LIN {X 0,Y 523.335,Z 404.353,A -85,B 0,C 180,E1 -4767.691,E2 -4767.691} C_VEL
LIN {X 0,Y 523.256,Z 405.957,A -85,B 0,C 180,E1 -4769.23,E2 -4769.23} C_VEL
LIN {X 0,Y 523.257,Z 406.174,A -85,B 0,C 180,E1 -4770,E2 -4770} C_VEL
LIN {X 0,Y 523.275,Z 405.351,A -85,B 0,C 180,E1 -4771.539,E2 -4771.539} C_VEL
LIN {X 0,Y 523.335,Z 404.357,A -85,B 0,C 180,E1 -4772.309,E2 -4772.309} C_VEL
LIN {X 0,Y 523.367,Z 402.961,A -85,B 0,C 180,E1 -4773.079,E2 -4773.079} C_VEL
LIN {X 0,Y 523.422,Z 400.024,A -85,B 0,C 180,E1 -4774.235,E2 -4774.235} C_VEL
LIN {X 0,Y 523.455,Z 396.045,A -85,B 0,C 180,E1 -4775.392,E2 -4775.392} C_VEL
LIN {X 0,Y 523.507,Z 389.976,A -85,B 0,C 180,E1 -4776.736,E2 -4776.736} C_VEL
LIN {X 0,Y 523.643,Z 383.242,A -85,B 0,C 180,E1 -4777.907,E2 -4777.907} C_VEL
LIN {X 0,Y 523.826,Z 374.948,A -85,B 0,C 180,E1 -4779.07,E2 -4779.07} C_VEL
LIN {X 0,Y 524.03,Z 366.449,A -85,B 0,C 180,E1 -4780.04,E2 -4780.04} C_VEL
LIN {X 0,Y 524.307,Z 355.951,A -85,B 0,C 180,E1 -4781.011,E2 -4781.011} C_VEL
LIN {X 0,Y 524.58,Z 345.751,A -85,B 0,C 180,E1 -4781.776,E2 -4781.776} C_VEL
LIN {X 0,Y 524.893,Z 334.187,A -85,B 0,C 180,E1 -4782.468,E2 -4782.468} C_VEL
LIN {X 0,Y 525.134,Z 322.52,A -85,B 0,C 180,E1 -4783.003,E2 -4783.003} C_VEL
LIN {X 0,Y 525.347,Z 309.079,A -85,B 0,C 180,E1 -4783.44,E2 -4783.44} C_VEL
LIN {X 0,Y 525.596,Z 295.824,A -85,B 0,C 180,E1 -4783.705,E2 -4783.705} C_VEL
LIN {X 0,Y 525.799,Z 203.654,A -85,B 0,C 180,E1 -4784.971,E2 -4784.971} C_VEL
LIN {X 0,Y 524.231,Z 193.19,A -85,B 0,C 180,E1 -4785.176,E2 -4785.176} C_VEL
LIN {X 0,Y 524.601,Z 174.823,A -85,B 0,C 180,E1 -4787.977,E2 -4787.977} C_VEL
LIN {X 0,Y 525.054,Z 155.376,A -85,B 0,C 180,E1 -4790.98,E2 -4790.98} C_VEL
LIN {X 0,Y 525.297,Z 140.922,A -85,B 0,C 180,E1 -4793.245,E2 -4793.245} C_VEL
LIN {X 0,Y 523.934,Z 133.223,A -85,B 0,C 180,E1 -4794.571,E2 -4794.571} C_VEL
LIN {X 0,Y 523.918,Z 133.225,A -85,B 0,C 180,E1 -4797.706,E2 -4797.706} C_VEL
LIN {X 0,Y 523.941,Z 133.217,A -85,B 0,C 180,E1 -4800.644,E2 -4800.644} C_VEL
LIN {X 0,Y 523.923,Z 133.224,A -85,B 0,C 180,E1 -4803.728,E2 -4803.728} C_VEL
LIN {X 0,Y 523.893,Z 133.222,A -85,B 0,C 180,E1 -4806.399,E2 -4806.399} C_VEL
LIN {X 0,Y 523.913,Z 133.224,A -85,B 0,C 180,E1 -4809.084,E2 -4809.084} C_VEL
LIN {X 0,Y 523.906,Z 133.22,A -85,B 0,C 180,E1 -4812.122,E2 -4812.122} C_VEL
LIN {X 0,Y 523.932,Z 133.224,A -85,B 0,C 180,E1 -4815.31,E2 -4815.31} C_VEL
LIN {X 0,Y 523.913,Z 133.222,A -85,B 0,C 180,E1 -4818.694,E2 -4818.694} C_VEL
LIN {X 0,Y 523.904,Z 133.22,A -85,B 0,C 180,E1 -4821.897,E2 -4821.897} C_VEL
LIN {X 0,Y 523.909,Z 133.228,A -85,B 0,C 180,E1 -4824.912,E2 -4824.912} C_VEL
LIN {X 0,Y 523.922,Z 133.218,A -85,B 0,C 180,E1 -4827.68,E2 -4827.68} C_VEL
LIN {X 0,Y 523.926,Z 133.225,A -85,B 0,C 180,E1 -4830.68,E2 -4830.68} C_VEL
LIN {X 0,Y 523.893,Z 133.222,A -85,B 0,C 180,E1 -4833.724,E2 -4833.724} C_VEL
LIN {X 0,Y 523.895,Z 133.225,A -85,B 0,C 180,E1 -4836.269,E2 -4836.269} C_VEL
LIN {X 0,Y 523.919,Z 133.224,A -85,B 0,C 180,E1 -4838.765,E2 -4838.765} C_VEL
LIN {X 0,Y 523.914,Z 133.22,A -85,B 0,C 180,E1 -4841.219,E2 -4841.219} C_VEL
LIN {X 0,Y 523.899,Z 133.229,A -85,B 0,C 180,E1 -4844.437,E2 -4844.437} C_VEL
LIN {X 0,Y 523.934,Z 133.217,A -85,B 0,C 180,E1 -4847.607,E2 -4847.607} C_VEL
LIN {X 0,Y 523.933,Z 133.219,A -85,B 0,C 180,E1 -4850.737,E2 -4850.737} C_VEL
LIN {X 0,Y 523.99,Z 133.214,A -85,B 0,C 180,E1 -4853.84,E2 -4853.84} C_VEL
LIN {X 0,Y 524.093,Z 133.201,A -85,B 0,C 180,E1 -4857.694,E2 -4857.694} C_VEL
LIN {X 0,Y 524.086,Z 133.206,A -85,B 0,C 180,E1 -4860,E2 -4860} C_VEL
LIN {X 0,Y 524.094,Z 133.2,A -85,B 0,C 180,E1 -4862.306,E2 -4862.306} C_VEL
LIN {X 0,Y 523.999,Z 133.212,A -85,B 0,C 180,E1 -4866.16,E2 -4866.16} C_VEL
LIN {X 0,Y 523.968,Z 133.215,A -85,B 0,C 180,E1 -4869.262,E2 -4869.262} C_VEL
LIN {X 0,Y 523.987,Z 133.218,A -85,B 0,C 180,E1 -4871.736,E2 -4871.736} C_VEL
LIN {X 0,Y 523.973,Z 133.214,A -85,B 0,C 180,E1 -4875.049,E2 -4875.049} C_VEL
LIN {X 0,Y 523.903,Z 133.223,A -85,B 0,C 180,E1 -4877.971,E2 -4877.971} C_VEL
LIN {X 0,Y 523.942,Z 133.215,A -85,B 0,C 180,E1 -4880.411,E2 -4880.411} C_VEL
LIN {X 0,Y 523.897,Z 133.224,A -85,B 0,C 180,E1 -4882.894,E2 -4882.894} C_VEL
LIN {X 0,Y 523.89,Z 133.229,A -85,B 0,C 180,E1 -4885.422,E2 -4885.422} C_VEL
LIN {X 0,Y 523.897,Z 133.221,A -85,B 0,C 180,E1 -4888.003,E2 -4888.003} C_VEL
LIN {X 0,Y 523.926,Z 133.223,A -85,B 0,C 180,E1 -4890.853,E2 -4890.853} C_VEL
LIN {X 0,Y 523.922,Z 133.219,A -85,B 0,C 180,E1 -4893.73,E2 -4893.73} C_VEL
LIN {X 0,Y 523.895,Z 133.223,A -85,B 0,C 180,E1 -4896.402,E2 -4896.402} C_VEL
LIN {X 0,Y 523.905,Z 133.226,A -85,B 0,C 180,E1 -4899.086,E2 -4899.086} C_VEL
LIN {X 0,Y 523.902,Z 133.221,A -85,B 0,C 180,E1 -4902.124,E2 -4902.124} C_VEL
LIN {X 0,Y 523.935,Z 133.218,A -85,B 0,C 180,E1 -4905.311,E2 -4905.311} C_VEL
LIN {X 0,Y 523.895,Z 133.227,A -85,B 0,C 180,E1 -4906.872,E2 -4906.872} C_VEL
LIN {X 0,Y 523.223,Z 133.308,A -85,B 0,C 180,E1 -4907.513,E2 -4907.513} C_VEL
LIN {X 0,Y 520.362,Z 133.67,A -85,B 0,C 180,E1 -4908.555,E2 -4908.555} C_VEL
LIN {X 0,Y 517.955,Z 133.965,A -85,B 0,C 180,E1 -4909.393,E2 -4909.393} C_VEL
LIN {X 0,Y 516.935,Z 134.091,A -85,B 0,C 180,E1 -4910.041,E2 -4910.041} C_VEL
LIN {X 0,Y 516.859,Z 134.102,A -85,B 0,C 180,E1 -4910.261,E2 -4910.261} C_VEL
LIN {X 0,Y 516.85,Z 134.099,A -85,B 0,C 180,E1 -4913.253,E2 -4913.253} C_VEL
LIN {X 0,Y 516.904,Z 134.097,A -85,B 0,C 180,E1 -4916.121,E2 -4916.121} C_VEL
LIN {X 0,Y 516.886,Z 134.096,A -85,B 0,C 180,E1 -4918.937,E2 -4918.937} C_VEL
LIN {X 0,Y 516.85,Z 134.1,A -85,B 0,C 180,E1 -4921.582,E2 -4921.582} C_VEL
LIN {X 0,Y 516.877,Z 134.104,A -85,B 0,C 180,E1 -4924.209,E2 -4924.209} C_VEL
LIN {X 0,Y 516.857,Z 134.099,A -85,B 0,C 180,E1 -4926.777,E2 -4926.777} C_VEL
LIN {X 0,Y 516.968,Z 134.097,A -85,B 0,C 180,E1 -4930.132,E2 -4930.132} C_VEL
LIN {X 0,Y 517.566,Z 139.303,A -85,B 0,C 180,E1 -4931.187,E2 -4931.187} C_VEL
LIN {X 0,Y 517.249,Z 154.128,A -85,B 0,C 180,E1 -4934.03,E2 -4934.03} C_VEL
LIN {X 0,Y 517.253,Z 157.604,A -85,B 0,C 180,E1 -4934.68,E2 -4934.68} C_VEL
LIN {X 0,Y 519.135,Z 167.747,A -85,B 0,C 180,E1 -4934.89,E2 -4934.89} C_VEL
LIN {X 0,Y 518.683,Z 264.861,A -85,B 0,C 180,E1 -4936.259,E2 -4936.259} C_VEL
LIN {X 0,Y 518.509,Z 278.018,A -85,B 0,C 180,E1 -4936.604,E2 -4936.604} C_VEL
LIN {X 0,Y 518.244,Z 291.213,A -85,B 0,C 180,E1 -4937.121,E2 -4937.121} C_VEL
LIN {X 0,Y 517.973,Z 303.019,A -85,B 0,C 180,E1 -4937.757,E2 -4937.757} C_VEL
LIN {X 0,Y 517.715,Z 314.443,A -85,B 0,C 180,E1 -4938.549,E2 -4938.549} C_VEL
LIN {X 0,Y 517.401,Z 324.683,A -85,B 0,C 180,E1 -4939.434,E2 -4939.434} C_VEL
LIN {X 0,Y 517.114,Z 333.868,A -85,B 0,C 180,E1 -4940.417,E2 -4940.417} C_VEL
LIN {X 0,Y 516.821,Z 342.781,A -85,B 0,C 180,E1 -4941.595,E2 -4941.595} C_VEL
LIN {X 0,Y 516.621,Z 349.955,A -85,B 0,C 180,E1 -4942.772,E2 -4942.772} C_VEL
LIN {X 0,Y 516.511,Z 356.489,A -85,B 0,C 180,E1 -4944.143,E2 -4944.143} C_VEL
LIN {X 0,Y 516.351,Z 360.813,A -85,B 0,C 180,E1 -4945.316,E2 -4945.316} C_VEL
LIN {X 0,Y 516.378,Z 363.097,A -85,B 0,C 180,E1 -4946.098,E2 -4946.098} C_VEL
LIN {X 0,Y 516.353,Z 364.958,A -85,B 0,C 180,E1 -4946.88,E2 -4946.88} C_VEL
LIN {X 0,Y 516.267,Z 366.366,A -85,B 0,C 180,E1 -4947.66,E2 -4947.66} C_VEL
LIN {X 0,Y 516.17,Z 367.982,A -85,B 0,C 180,E1 -4949.22,E2 -4949.22} C_VEL
LIN {X 0,Y 516.167,Z 368.219,A -85,B 0,C 180,E1 -4950,E2 -4950} C_VEL
LIN {X 0,Y 516.17,Z 368.036,A -85,B 0,C 180,E1 -4950.781,E2 -4950.781} C_VEL
LIN {X 0,Y 516.267,Z 366.49,A -85,B 0,C 180,E1 -4952.341,E2 -4952.341} C_VEL
LIN {X 0,Y 516.354,Z 365.137,A -85,B 0,C 180,E1 -4953.121,E2 -4953.121} C_VEL
LIN {X 0,Y 516.394,Z 362.28,A -85,B 0,C 180,E1 -4954.293,E2 -4954.293} C_VEL
LIN {X 0,Y 516.409,Z 358.408,A -85,B 0,C 180,E1 -4955.467,E2 -4955.467} C_VEL
LIN {X 0,Y 516.552,Z 352.462,A -85,B 0,C 180,E1 -4956.834,E2 -4956.834} C_VEL
LIN {X 0,Y 516.747,Z 345.894,A -85,B 0,C 180,E1 -4958.014,E2 -4958.014} C_VEL
LIN {X 0,Y 516.944,Z 337.759,A -85,B 0,C 180,E1 -4959.192,E2 -4959.192} C_VEL
LIN {X 0,Y 517.207,Z 329.428,A -85,B 0,C 180,E1 -4960.175,E2 -4960.175} C_VEL
LIN {X 0,Y 517.563,Z 319.139,A -85,B 0,C 180,E1 -4961.157,E2 -4961.157} C_VEL
LIN {X 0,Y 517.858,Z 307.684,A -85,B 0,C 180,E1 -4962.033,E2 -4962.033} C_VEL
LIN {X 0,Y 518.157,Z 295.983,A -85,B 0,C 180,E1 -4962.733,E2 -4962.733} C_VEL
LIN {X 0,Y 518.422,Z 283.972,A -85,B 0,C 180,E1 -4963.275,E2 -4963.275} C_VEL
LIN {X 0,Y 518.639,Z 270.9,A -85,B 0,C 180,E1 -4963.693,E2 -4963.693} C_VEL
LIN {X 0,Y 518.798,Z 258.393,A -85,B 0,C 180,E1 -4963.939,E2 -4963.939} C_VEL
LIN {X 0,Y 519.01,Z 167.183,A -85,B 0,C 180,E1 -4965.211,E2 -4965.211} C_VEL
LIN {X 0,Y 517.227,Z 157.657,A -85,B 0,C 180,E1 -4965.401,E2 -4965.401} C_VEL
LIN {X 0,Y 517.506,Z 141.844,A -85,B 0,C 180,E1 -4968.406,E2 -4968.406} C_VEL
LIN {X 0,Y 517.481,Z 137.669,A -85,B 0,C 180,E1 -4969.229,E2 -4969.229} C_VEL
LIN {X 0,Y 516.97,Z 134.093,A -85,B 0,C 180,E1 -4969.968,E2 -4969.968} C_VEL
LIN {X 0,Y 516.86,Z 134.099,A -85,B 0,C 180,E1 -4973.224,E2 -4973.224} C_VEL
LIN {X 0,Y 516.897,Z 134.099,A -85,B 0,C 180,E1 -4976.185,E2 -4976.185} C_VEL
LIN {X 0,Y 516.921,Z 134.092,A -85,B 0,C 180,E1 -4979.305,E2 -4979.305} C_VEL
LIN {X 0,Y 516.897,Z 134.093,A -85,B 0,C 180,E1 -4982.543,E2 -4982.543} C_VEL
LIN {X 0,Y 516.865,Z 134.101,A -85,B 0,C 180,E1 -4985.329,E2 -4985.329} C_VEL
LIN {X 0,Y 516.878,Z 134.099,A -85,B 0,C 180,E1 -4987.942,E2 -4987.942} C_VEL
LIN {X 0,Y 516.864,Z 134.098,A -85,B 0,C 180,E1 -4990.743,E2 -4990.743} C_VEL
LIN {X 0,Y 516.859,Z 134.099,A -85,B 0,C 180,E1 -4992.834,E2 -4992.834} C_VEL
LIN {X 0,Y 516.895,Z 134.097,A -85,B 0,C 180,E1 -4995.007,E2 -4995.007} C_VEL
LIN {X 0,Y 516.901,Z 134.093,A -85,B 0,C 180,E1 -4998.4,E2 -4998.4} C_VEL
LIN {X 0,Y 516.875,Z 134.103,A -85,B 0,C 180,E1 -5001.283,E2 -5001.283} C_VEL
LIN {X 0,Y 516.864,Z 134.097,A -85,B 0,C 180,E1 -5004.219,E2 -5004.219} C_VEL
LIN {X 0,Y 516.877,Z 134.104,A -85,B 0,C 180,E1 -5007.052,E2 -5007.052} C_VEL
LIN {X 0,Y 516.86,Z 134.098,A -85,B 0,C 180,E1 -5009.794,E2 -5009.794} C_VEL
LIN {X 0,Y 516.879,Z 134.099,A -85,B 0,C 180,E1 -5012.464,E2 -5012.464} C_VEL
LIN {X 0,Y 516.848,Z 134.104,A -85,B 0,C 180,E1 -5015.068,E2 -5015.068} C_VEL
LIN {X 0,Y 516.867,Z 134.097,A -85,B 0,C 180,E1 -5017.621,E2 -5017.621} C_VEL
LIN {X 0,Y 516.915,Z 134.093,A -85,B 0,C 180,E1 -5020.129,E2 -5020.129} C_VEL
LIN {X 0,Y 516.861,Z 134.106,A -85,B 0,C 180,E1 -5022.594,E2 -5022.594} C_VEL
LIN {X 0,Y 516.928,Z 134.091,A -85,B 0,C 180,E1 -5025.03,E2 -5025.03} C_VEL
LIN {X 0,Y 516.963,Z 134.091,A -85,B 0,C 180,E1 -5028.234,E2 -5028.234} C_VEL
LIN {X 0,Y 516.925,Z 134.09,A -85,B 0,C 180,E1 -5031.399,E2 -5031.399} C_VEL
LIN {X 0,Y 516.976,Z 134.088,A -85,B 0,C 180,E1 -5034.539,E2 -5034.539} C_VEL
LIN {X 0,Y 517.068,Z 134.074,A -85,B 0,C 180,E1 -5037.663,E2 -5037.663} C_VEL
LIN {X 0,Y 517.06,Z 134.081,A -85,B 0,C 180,E1 -5040,E2 -5040} C_VEL
LIN {X 0,Y 517.068,Z 134.076,A -85,B 0,C 180,E1 -5042.337,E2 -5042.337} C_VEL
LIN {X 0,Y 516.962,Z 134.089,A -85,B 0,C 180,E1 -5046.244,E2 -5046.244} C_VEL
LIN {X 0,Y 516.9,Z 134.096,A -85,B 0,C 180,E1 -5049.39,E2 -5049.39} C_VEL
LIN {X 0,Y 516.875,Z 134.096,A -85,B 0,C 180,E1 -5052.565,E2 -5052.565} C_VEL
LIN {X 0,Y 516.879,Z 134.097,A -85,B 0,C 180,E1 -5055.121,E2 -5055.121} C_VEL
LIN {X 0,Y 516.865,Z 134.098,A -85,B 0,C 180,E1 -5058.224,E2 -5058.224} C_VEL
LIN {X 0,Y 516.867,Z 134.097,A -85,B 0,C 180,E1 -5060.703,E2 -5060.703} C_VEL
LIN {X 0,Y 516.836,Z 134.107,A -85,B 0,C 180,E1 -5063.225,E2 -5063.225} C_VEL
LIN {X 0,Y 516.875,Z 134.096,A -85,B 0,C 180,E1 -5066.181,E2 -5066.181} C_VEL
LIN {X 0,Y 516.825,Z 134.102,A -85,B 0,C 180,E1 -5068.421,E2 -5068.421} C_VEL
LIN {X 0,Y 516.845,Z 134.107,A -85,B 0,C 180,E1 -5071.113,E2 -5071.113} C_VEL
LIN {X 0,Y 516.878,Z 134.096,A -85,B 0,C 180,E1 -5073.962,E2 -5073.962} C_VEL
LIN {X 0,Y 516.847,Z 134.104,A -85,B 0,C 180,E1 -5076.749,E2 -5076.749} C_VEL
LIN {X 0,Y 516.856,Z 134.099,A -85,B 0,C 180,E1 -5079.724,E2 -5079.724} C_VEL
LIN {X 0,Y 516.841,Z 134.109,A -85,B 0,C 180,E1 -5082.836,E2 -5082.836} C_VEL
LIN {X 0,Y 516.895,Z 134.099,A -85,B 0,C 180,E1 -5085.007,E2 -5085.007} C_VEL
LIN {X 0,Y 516.855,Z 134.103,A -85,B 0,C 180,E1 -5088.406,E2 -5088.406} C_VEL
LIN {X 0,Y 516.876,Z 134.097,A -85,B 0,C 180,E1 -5091.284,E2 -5091.284} C_VEL
LIN {X 0,Y 516.865,Z 134.101,A -85,B 0,C 180,E1 -5094.219,E2 -5094.219} C_VEL
LIN {X 0,Y 516.881,Z 134.097,A -85,B 0,C 180,E1 -5097.052,E2 -5097.052} C_VEL
LIN {X 0,Y 516.868,Z 134.1,A -85,B 0,C 180,E1 -5099.795,E2 -5099.795} C_VEL
LIN {X 0,Y 516.878,Z 134.104,A -85,B 0,C 180,E1 -5102.464,E2 -5102.464} C_VEL
LIN {X 0,Y 516.886,Z 134.117,A -85,B 0,C 180,E1 -5105.299,E2 -5105.299} C_VEL
LIN {X 0,Y 518.432,Z 143.303,A -85,B 0,C 180,E1 -5106.85,E2 -5106.85} C_VEL
LIN {X 0,Y 518.002,Z 160.237,A -85,B 0,C 180,E1 -5109.531,E2 -5109.531} C_VEL
LIN {X 0,Y 517.536,Z 178.843,A -85,B 0,C 180,E1 -5112.436,E2 -5112.436} C_VEL
LIN {X 0,Y 517.219,Z 192.958,A -85,B 0,C 180,E1 -5114.618,E2 -5114.618} C_VEL
LIN {X 0,Y 519.015,Z 206.166,A -85,B 0,C 180,E1 -5114.868,E2 -5114.868} C_VEL
LIN {X 0,Y 518.64,Z 301.382,A -85,B 0,C 180,E1 -5116.207,E2 -5116.207} C_VEL
LIN {X 0,Y 518.37,Z 314.674,A -85,B 0,C 180,E1 -5116.549,E2 -5116.549} C_VEL
LIN {X 0,Y 518.043,Z 327.977,A -85,B 0,C 180,E1 -5117.065,E2 -5117.065} C_VEL
LIN {X 0,Y 517.77,Z 339.847,A -85,B 0,C 180,E1 -5117.7,E2 -5117.7} C_VEL
LIN {X 0,Y 517.516,Z 350.763,A -85,B 0,C 180,E1 -5118.445,E2 -5118.445} C_VEL
LIN {X 0,Y 517.201,Z 361.222,A -85,B 0,C 180,E1 -5119.33,E2 -5119.33} C_VEL
LIN {X 0,Y 516.926,Z 369.774,A -85,B 0,C 180,E1 -5120.215,E2 -5120.215} C_VEL
LIN {X 0,Y 516.694,Z 377.667,A -85,B 0,C 180,E1 -5121.198,E2 -5121.198} C_VEL
LIN {X 0,Y 516.532,Z 385.378,A -85,B 0,C 180,E1 -5122.376,E2 -5122.376} C_VEL
LIN {X 0,Y 516.376,Z 392.487,A -85,B 0,C 180,E1 -5123.749,E2 -5123.749} C_VEL
LIN {X 0,Y 516.312,Z 397.217,A -85,B 0,C 180,E1 -5124.924,E2 -5124.924} C_VEL
LIN {X 0,Y 516.352,Z 400.834,A -85,B 0,C 180,E1 -5126.097,E2 -5126.097} C_VEL
LIN {X 0,Y 516.282,Z 402.697,A -85,B 0,C 180,E1 -5126.878,E2 -5126.878} C_VEL
LIN {X 0,Y 516.261,Z 404.094,A -85,B 0,C 180,E1 -5127.659,E2 -5127.659} C_VEL
LIN {X 0,Y 516.166,Z 405.698,A -85,B 0,C 180,E1 -5129.219,E2 -5129.219} C_VEL
LIN {X 0,Y 516.164,Z 405.915,A -85,B 0,C 180,E1 -5130,E2 -5130} C_VEL
LIN {X 0,Y 516.192,Z 405.092,A -85,B 0,C 180,E1 -5131.56,E2 -5131.56} C_VEL
LIN {X 0,Y 516.261,Z 404.099,A -85,B 0,C 180,E1 -5132.34,E2 -5132.34} C_VEL
LIN {X 0,Y 516.282,Z 402.702,A -85,B 0,C 180,E1 -5133.121,E2 -5133.121} C_VEL
LIN {X 0,Y 516.31,Z 399.763,A -85,B 0,C 180,E1 -5134.293,E2 -5134.293} C_VEL
LIN {X 0,Y 516.367,Z 395.785,A -85,B 0,C 180,E1 -5135.467,E2 -5135.467} C_VEL
LIN {X 0,Y 516.411,Z 390.616,A -85,B 0,C 180,E1 -5136.653,E2 -5136.653} C_VEL
LIN {X 0,Y 516.543,Z 384.22,A -85,B 0,C 180,E1 -5137.819,E2 -5137.819} C_VEL
LIN {X 0,Y 516.748,Z 376.181,A -85,B 0,C 180,E1 -5138.998,E2 -5138.998} C_VEL
LIN {X 0,Y 516.952,Z 367.991,A -85,B 0,C 180,E1 -5139.981,E2 -5139.981} C_VEL
LIN {X 0,Y 517.289,Z 358.008,A -85,B 0,C 180,E1 -5140.964,E2 -5140.964} C_VEL
LIN {X 0,Y 517.58,Z 348.163,A -85,B 0,C 180,E1 -5141.752,E2 -5141.752} C_VEL
LIN {X 0,Y 517.845,Z 337.067,A -85,B 0,C 180,E1 -5142.464,E2 -5142.464} C_VEL
LIN {X 0,Y 518.152,Z 324.601,A -85,B 0,C 180,E1 -5143.081,E2 -5143.081} C_VEL
LIN {X 0,Y 518.424,Z 311.567,A -85,B 0,C 180,E1 -5143.548,E2 -5143.548} C_VEL
LIN {X 0,Y 518.672,Z 298.583,A -85,B 0,C 180,E1 -5143.841,E2 -5143.841} C_VEL
LIN {X 0,Y 518.978,Z 204.566,A -85,B 0,C 180,E1 -5145.156,E2 -5145.156} C_VEL
LIN {X 0,Y 517.228,Z 192.912,A -85,B 0,C 180,E1 -5145.39,E2 -5145.39} C_VEL
LIN {X 0,Y 517.633,Z 174.779,A -85,B 0,C 180,E1 -5148.196,E2 -5148.196} C_VEL
LIN {X 0,Y 518.163,Z 153.812,A -85,B 0,C 180,E1 -5151.481,E2 -5151.481} C_VEL
LIN {X 0,Y 518.344,Z 141.985,A -85,B 0,C 180,E1 -5153.364,E2 -5153.364} C_VEL
LIN {X 0,Y 516.891,Z 134.1,A -85,B 0,C 180,E1 -5154.739,E2 -5154.739} C_VEL
LIN {X 0,Y 516.876,Z 134.102,A -85,B 0,C 180,E1 -5157.535,E2 -5157.535} C_VEL
LIN {X 0,Y 516.864,Z 134.101,A -85,B 0,C 180,E1 -5160.205,E2 -5160.205} C_VEL
LIN {X 0,Y 516.877,Z 134.097,A -85,B 0,C 180,E1 -5162.947,E2 -5162.947} C_VEL
LIN {X 0,Y 516.862,Z 134.102,A -85,B 0,C 180,E1 -5165.78,E2 -5165.78} C_VEL
LIN {X 0,Y 516.873,Z 134.097,A -85,B 0,C 180,E1 -5168.715,E2 -5168.715} C_VEL
LIN {X 0,Y 516.879,Z 134.098,A -85,B 0,C 180,E1 -5171.777,E2 -5171.777} C_VEL
LIN {X 0,Y 516.89,Z 134.1,A -85,B 0,C 180,E1 -5175.006,E2 -5175.006} C_VEL
LIN {X 0,Y 516.849,Z 134.1,A -85,B 0,C 180,E1 -5178.405,E2 -5178.405} C_VEL
LIN {X 0,Y 516.868,Z 134.102,A -85,B 0,C 180,E1 -5181.283,E2 -5181.283} C_VEL
LIN {X 0,Y 516.857,Z 134.099,A -85,B 0,C 180,E1 -5184.218,E2 -5184.218} C_VEL
LIN {X 0,Y 516.871,Z 134.103,A -85,B 0,C 180,E1 -5187.051,E2 -5187.051} C_VEL
LIN {X 0,Y 516.853,Z 134.098,A -85,B 0,C 180,E1 -5189.794,E2 -5189.794} C_VEL
LIN {X 0,Y 516.865,Z 134.102,A -85,B 0,C 180,E1 -5192.464,E2 -5192.464} C_VEL
LIN {X 0,Y 516.835,Z 134.104,A -85,B 0,C 180,E1 -5195.068,E2 -5195.068} C_VEL
LIN {X 0,Y 516.86,Z 134.098,A -85,B 0,C 180,E1 -5197.621,E2 -5197.621} C_VEL
LIN {X 0,Y 516.903,Z 134.096,A -85,B 0,C 180,E1 -5200.129,E2 -5200.129} C_VEL
LIN {X 0,Y 516.854,Z 134.105,A -85,B 0,C 180,E1 -5202.594,E2 -5202.594} C_VEL
LIN {X 0,Y 516.921,Z 134.091,A -85,B 0,C 180,E1 -5205.029,E2 -5205.029} C_VEL
LIN {X 0,Y 516.914,Z 134.099,A -85,B 0,C 180,E1 -5208.232,E2 -5208.232} C_VEL
LIN {X 0,Y 516.908,Z 134.092,A -85,B 0,C 180,E1 -5211.399,E2 -5211.399} C_VEL
LIN {X 0,Y 516.969,Z 134.087,A -85,B 0,C 180,E1 -5214.539,E2 -5214.539} C_VEL
LIN {X 0,Y 517.062,Z 134.076,A -85,B 0,C 180,E1 -5217.663,E2 -5217.663} C_VEL
LIN {X 0,Y 517.054,Z 134.082,A -85,B 0,C 180,E1 -5220,E2 -5220} C_VEL
LIN {X 0,Y 517.063,Z 134.075,A -85,B 0,C 180,E1 -5222.337,E2 -5222.337} C_VEL
LIN {X 0,Y 516.964,Z 134.087,A -85,B 0,C 180,E1 -5226.244,E2 -5226.244} C_VEL
LIN {X 0,Y 516.924,Z 134.094,A -85,B 0,C 180,E1 -5229.39,E2 -5229.39} C_VEL
LIN {X 0,Y 516.942,Z 134.094,A -85,B 0,C 180,E1 -5231.807,E2 -5231.807} C_VEL
LIN {X 0,Y 516.926,Z 134.093,A -85,B 0,C 180,E1 -5235.143,E2 -5235.143} C_VEL
LIN {X 0,Y 516.866,Z 134.097,A -85,B 0,C 180,E1 -5238.224,E2 -5238.224} C_VEL
LIN {X 0,Y 516.892,Z 134.095,A -85,B 0,C 180,E1 -5240.702,E2 -5240.702} C_VEL
LIN {X 0,Y 516.846,Z 134.107,A -85,B 0,C 180,E1 -5243.225,E2 -5243.225} C_VEL
LIN {X 0,Y 516.872,Z 134.096,A -85,B 0,C 180,E1 -5246.183,E2 -5246.183} C_VEL
LIN {X 0,Y 516.894,Z 134.1,A -85,B 0,C 180,E1 -5249.306,E2 -5249.306} C_VEL
LIN {X 0,Y 516.885,Z 134.097,A -85,B 0,C 180,E1 -5252.544,E2 -5252.544} C_VEL
LIN {X 0,Y 516.857,Z 134.102,A -85,B 0,C 180,E1 -5255.33,E2 -5255.33} C_VEL
LIN {X 0,Y 516.871,Z 134.096,A -85,B 0,C 180,E1 -5257.943,E2 -5257.943} C_VEL
LIN {X 0,Y 516.847,Z 134.107,A -85,B 0,C 180,E1 -5260.745,E2 -5260.745} C_VEL
LIN {X 0,Y 516.875,Z 134.096,A -85,B 0,C 180,E1 -5263.904,E2 -5263.904} C_VEL
LIN {X 0,Y 516.842,Z 134.1,A -85,B 0,C 180,E1 -5266.873,E2 -5266.873} C_VEL
LIN {X 0,Y 516.876,Z 134.096,A -85,B 0,C 180,E1 -5269.591,E2 -5269.591} C_VEL
LIN {X 0,Y 516.859,Z 134.102,A -85,B 0,C 180,E1 -5270.261,E2 -5270.261} C_VEL
LIN {X 0,Y 516.212,Z 134.188,A -85,B 0,C 180,E1 -5270.911,E2 -5270.911} C_VEL
LIN {X 0,Y 513.365,Z 134.54,A -85,B 0,C 180,E1 -5271.966,E2 -5271.966} C_VEL
LIN {X 0,Y 510.941,Z 134.839,A -85,B 0,C 180,E1 -5272.816,E2 -5272.816} C_VEL
LIN {X 0,Y 509.892,Z 134.966,A -85,B 0,C 180,E1 -5273.473,E2 -5273.473} C_VEL
LIN {X 0,Y 509.804,Z 134.977,A -85,B 0,C 180,E1 -5273.695,E2 -5273.695} C_VEL
LIN {X 0,Y 509.856,Z 134.977,A -85,B 0,C 180,E1 -5276.54,E2 -5276.54} C_VEL
LIN {X 0,Y 509.832,Z 134.973,A -85,B 0,C 180,E1 -5279.334,E2 -5279.334} C_VEL
LIN {X 0,Y 509.835,Z 134.979,A -85,B 0,C 180,E1 -5282.052,E2 -5282.052} C_VEL
LIN {X 0,Y 509.805,Z 134.978,A -85,B 0,C 180,E1 -5284.701,E2 -5284.701} C_VEL
LIN {X 0,Y 509.825,Z 134.975,A -85,B 0,C 180,E1 -5287.459,E2 -5287.459} C_VEL
LIN {X 0,Y 509.94,Z 135.08,A -85,B 0,C 180,E1 -5290.03,E2 -5290.03} C_VEL
LIN {X 0,Y 510.594,Z 140.443,A -85,B 0,C 180,E1 -5291.128,E2 -5291.128} C_VEL
LIN {X 0,Y 510.248,Z 155.397,A -85,B 0,C 180,E1 -5294.01,E2 -5294.01} C_VEL
LIN {X 0,Y 510.245,Z 157.828,A -85,B 0,C 180,E1 -5294.467,E2 -5294.467} C_VEL
LIN {X 0,Y 512.314,Z 169.462,A -85,B 0,C 180,E1 -5294.705,E2 -5294.705} C_VEL
LIN {X 0,Y 511.813,Z 265.147,A -85,B 0,C 180,E1 -5296.071,E2 -5296.071} C_VEL
LIN {X 0,Y 511.611,Z 278.296,A -85,B 0,C 180,E1 -5296.42,E2 -5296.42} C_VEL
LIN {X 0,Y 511.325,Z 291.486,A -85,B 0,C 180,E1 -5296.943,E2 -5296.943} C_VEL
LIN {X 0,Y 511.022,Z 303.813,A -85,B 0,C 180,E1 -5297.621,E2 -5297.621} C_VEL
LIN {X 0,Y 510.777,Z 314.71,A -85,B 0,C 180,E1 -5298.392,E2 -5298.392} C_VEL
LIN {X 0,Y 510.427,Z 324.948,A -85,B 0,C 180,E1 -5299.288,E2 -5299.288} C_VEL
LIN {X 0,Y 510.098,Z 334.133,A -85,B 0,C 180,E1 -5300.284,E2 -5300.284} C_VEL
LIN {X 0,Y 509.81,Z 343.044,A -85,B 0,C 180,E1 -5301.478,E2 -5301.478} C_VEL
LIN {X 0,Y 509.581,Z 350.217,A -85,B 0,C 180,E1 -5302.671,E2 -5302.671} C_VEL
LIN {X 0,Y 509.474,Z 355.056,A -85,B 0,C 180,E1 -5303.665,E2 -5303.665} C_VEL
LIN {X 0,Y 509.264,Z 359.761,A -85,B 0,C 180,E1 -5304.854,E2 -5304.854} C_VEL
LIN {X 0,Y 509.312,Z 363.357,A -85,B 0,C 180,E1 -5306.044,E2 -5306.044} C_VEL
LIN {X 0,Y 509.265,Z 365.219,A -85,B 0,C 180,E1 -5306.836,E2 -5306.836} C_VEL
LIN {X 0,Y 509.198,Z 366.625,A -85,B 0,C 180,E1 -5307.627,E2 -5307.627} C_VEL
LIN {X 0,Y 509.083,Z 368.241,A -85,B 0,C 180,E1 -5309.209,E2 -5309.209} C_VEL
LIN {X 0,Y 509.078,Z 368.478,A -85,B 0,C 180,E1 -5310,E2 -5310} C_VEL
LIN {X 0,Y 509.082,Z 368.294,A -85,B 0,C 180,E1 -5310.791,E2 -5310.791} C_VEL
LIN {X 0,Y 509.198,Z 366.747,A -85,B 0,C 180,E1 -5312.373,E2 -5312.373} C_VEL
LIN {X 0,Y 509.266,Z 365.395,A -85,B 0,C 180,E1 -5313.165,E2 -5313.165} C_VEL
LIN {X 0,Y 509.322,Z 362.538,A -85,B 0,C 180,E1 -5314.353,E2 -5314.353} C_VEL
LIN {X 0,Y 509.356,Z 358.665,A -85,B 0,C 180,E1 -5315.543,E2 -5315.543} C_VEL
LIN {X 0,Y 509.491,Z 352.93,A -85,B 0,C 180,E1 -5316.887,E2 -5316.887} C_VEL
LIN {X 0,Y 509.7,Z 346.15,A -85,B 0,C 180,E1 -5318.125,E2 -5318.125} C_VEL
LIN {X 0,Y 509.94,Z 338.013,A -85,B 0,C 180,E1 -5319.32,E2 -5319.32} C_VEL
LIN {X 0,Y 510.212,Z 329.682,A -85,B 0,C 180,E1 -5320.316,E2 -5320.316} C_VEL
LIN {X 0,Y 510.586,Z 319.392,A -85,B 0,C 180,E1 -5321.312,E2 -5321.312} C_VEL
LIN {X 0,Y 510.895,Z 308.631,A -85,B 0,C 180,E1 -5322.15,E2 -5322.15} C_VEL
LIN {X 0,Y 511.225,Z 298.043,A -85,B 0,C 180,E1 -5322.808,E2 -5322.808} C_VEL
LIN {X 0,Y 511.49,Z 286.735,A -85,B 0,C 180,E1 -5323.357,E2 -5323.357} C_VEL
LIN {X 0,Y 511.695,Z 274.793,A -85,B 0,C 180,E1 -5323.781,E2 -5323.781} C_VEL
LIN {X 0,Y 511.879,Z 261.678,A -85,B 0,C 180,E1 -5324.08,E2 -5324.08} C_VEL
LIN {X 0,Y 512.196,Z 167.979,A -85,B 0,C 180,E1 -5325.41,E2 -5325.41} C_VEL
LIN {X 0,Y 510.245,Z 157.86,A -85,B 0,C 180,E1 -5325.617,E2 -5325.617} C_VEL
LIN {X 0,Y 510.529,Z 143.003,A -85,B 0,C 180,E1 -5328.459,E2 -5328.459} C_VEL
LIN {X 0,Y 510.504,Z 138.797,A -85,B 0,C 180,E1 -5329.293,E2 -5329.293} C_VEL
LIN {X 0,Y 509.927,Z 134.97,A -85,B 0,C 180,E1 -5330.102,E2 -5330.102} C_VEL
LIN {X 0,Y 509.821,Z 134.978,A -85,B 0,C 180,E1 -5333.564,E2 -5333.564} C_VEL
LIN {X 0,Y 509.873,Z 134.971,A -85,B 0,C 180,E1 -5336.369,E2 -5336.369} C_VEL
LIN {X 0,Y 509.86,Z 134.978,A -85,B 0,C 180,E1 -5339.726,E2 -5339.726} C_VEL
LIN {X 0,Y 509.875,Z 134.968,A -85,B 0,C 180,E1 -5342.774,E2 -5342.774} C_VEL
LIN {X 0,Y 509.824,Z 134.982,A -85,B 0,C 180,E1 -5345.578,E2 -5345.578} C_VEL
LIN {X 0,Y 509.848,Z 134.972,A -85,B 0,C 180,E1 -5348.338,E2 -5348.338} C_VEL
LIN {X 0,Y 509.845,Z 134.98,A -85,B 0,C 180,E1 -5351.426,E2 -5351.426} C_VEL
LIN {X 0,Y 509.839,Z 134.973,A -85,B 0,C 180,E1 -5354.67,E2 -5354.67} C_VEL
LIN {X 0,Y 509.844,Z 134.972,A -85,B 0,C 180,E1 -5358.105,E2 -5358.105} C_VEL
LIN {X 0,Y 509.831,Z 134.975,A -85,B 0,C 180,E1 -5360.646,E2 -5360.646} C_VEL
LIN {X 0,Y 509.807,Z 134.978,A -85,B 0,C 180,E1 -5363.645,E2 -5363.645} C_VEL
LIN {X 0,Y 509.837,Z 134.975,A -85,B 0,C 180,E1 -5366.537,E2 -5366.537} C_VEL
LIN {X 0,Y 509.825,Z 134.978,A -85,B 0,C 180,E1 -5369.333,E2 -5369.333} C_VEL
LIN {X 0,Y 509.832,Z 134.973,A -85,B 0,C 180,E1 -5372.051,E2 -5372.051} C_VEL
LIN {X 0,Y 509.806,Z 134.984,A -85,B 0,C 180,E1 -5374.7,E2 -5374.7} C_VEL
LIN {X 0,Y 509.822,Z 134.975,A -85,B 0,C 180,E1 -5377.459,E2 -5377.459} C_VEL
LIN {X 0,Y 509.904,Z 134.965,A -85,B 0,C 180,E1 -5379.844,E2 -5379.844} C_VEL
LIN {X 0,Y 509.843,Z 134.977,A -85,B 0,C 180,E1 -5382.346,E2 -5382.346} C_VEL
LIN {X 0,Y 509.881,Z 134.972,A -85,B 0,C 180,E1 -5384.818,E2 -5384.818} C_VEL
LIN {X 0,Y 509.898,Z 134.97,A -85,B 0,C 180,E1 -5388.124,E2 -5388.124} C_VEL
LIN {X 0,Y 509.88,Z 134.967,A -85,B 0,C 180,E1 -5391.279,E2 -5391.279} C_VEL
LIN {X 0,Y 509.912,Z 134.965,A -85,B 0,C 180,E1 -5393.67,E2 -5393.67} C_VEL
LIN {X 0,Y 509.881,Z 134.968,A -85,B 0,C 180,E1 -5396.839,E2 -5396.839} C_VEL
LIN {X 0,Y 509.918,Z 134.967,A -85,B 0,C 180,E1 -5398.42,E2 -5398.42} C_VEL
LIN {X 0,Y 510.029,Z 134.956,A -85,B 0,C 180,E1 -5400,E2 -5400} C_VEL
LIN {X 0,Y 510.036,Z 134.952,A -85,B 0,C 180,E1 -5402.369,E2 -5402.369} C_VEL
LIN {X 0,Y 509.929,Z 134.965,A -85,B 0,C 180,E1 -5405.536,E2 -5405.536} C_VEL
LIN {X 0,Y 509.87,Z 134.976,A -85,B 0,C 180,E1 -5407.923,E2 -5407.923} C_VEL
LIN {X 0,Y 509.855,Z 134.972,A -85,B 0,C 180,E1 -5411.127,E2 -5411.127} C_VEL
LIN {X 0,Y 509.811,Z 134.983,A -85,B 0,C 180,E1 -5413.554,E2 -5413.554} C_VEL
LIN {X 0,Y 509.787,Z 134.982,A -85,B 0,C 180,E1 -5416.005,E2 -5416.005} C_VEL
LIN {X 0,Y 509.822,Z 134.975,A -85,B 0,C 180,E1 -5418.485,E2 -5418.485} C_VEL
LIN {X 0,Y 509.813,Z 134.978,A -85,B 0,C 180,E1 -5421.003,E2 -5421.003} C_VEL
LIN {X 0,Y 509.798,Z 134.984,A -85,B 0,C 180,E1 -5423.565,E2 -5423.565} C_VEL
LIN {X 0,Y 509.811,Z 134.976,A -85,B 0,C 180,E1 -5426.356,E2 -5426.356} C_VEL
LIN {X 0,Y 509.789,Z 134.982,A -85,B 0,C 180,E1 -5428.85,E2 -5428.85} C_VEL
LIN {X 0,Y 509.793,Z 134.981,A -85,B 0,C 180,E1 -5431.592,E2 -5431.592} C_VEL
LIN {X 0,Y 509.831,Z 134.974,A -85,B 0,C 180,E1 -5434.415,E2 -5434.415} C_VEL
LIN {X 0,Y 509.804,Z 134.981,A -85,B 0,C 180,E1 -5437.342,E2 -5437.342} C_VEL
LIN {X 0,Y 509.812,Z 134.978,A -85,B 0,C 180,E1 -5440.385,E2 -5440.385} C_VEL
LIN {X 0,Y 509.804,Z 134.977,A -85,B 0,C 180,E1 -5443.574,E2 -5443.574} C_VEL
LIN {X 0,Y 509.805,Z 134.981,A -85,B 0,C 180,E1 -5446.427,E2 -5446.427} C_VEL
LIN {X 0,Y 509.813,Z 134.976,A -85,B 0,C 180,E1 -5449.616,E2 -5449.616} C_VEL
LIN {X 0,Y 509.807,Z 134.984,A -85,B 0,C 180,E1 -5452.658,E2 -5452.658} C_VEL
LIN {X 0,Y 509.839,Z 134.973,A -85,B 0,C 180,E1 -5455.801,E2 -5455.801} C_VEL
LIN {X 0,Y 509.845,Z 134.978,A -85,B 0,C 180,E1 -5458.721,E2 -5458.721} C_VEL
LIN {X 0,Y 509.839,Z 134.975,A -85,B 0,C 180,E1 -5461.153,E2 -5461.153} C_VEL
LIN {X 0,Y 509.852,Z 134.978,A -85,B 0,C 180,E1 -5463.826,E2 -5463.826} C_VEL
LIN {X 0,Y 509.856,Z 135.056,A -85,B 0,C 180,E1 -5465.133,E2 -5465.133} C_VEL
LIN {X 0,Y 511.367,Z 143.046,A -85,B 0,C 180,E1 -5466.512,E2 -5466.512} C_VEL
LIN {X 0,Y 511.284,Z 152.246,A -85,B 0,C 180,E1 -5468.002,E2 -5468.002} C_VEL
LIN {X 0,Y 510.748,Z 170.595,A -85,B 0,C 180,E1 -5470.925,E2 -5470.925} C_VEL
LIN {X 0,Y 510.272,Z 190.202,A -85,B 0,C 180,E1 -5474.01,E2 -5474.01} C_VEL
LIN {X 0,Y 510.227,Z 192.726,A -85,B 0,C 180,E1 -5474.405,E2 -5474.405} C_VEL
LIN {X 0,Y 512.168,Z 207.178,A -85,B 0,C 180,E1 -5474.678,E2 -5474.678} C_VEL
LIN {X 0,Y 511.758,Z 301.123,A -85,B 0,C 180,E1 -5476.018,E2 -5476.018} C_VEL
LIN {X 0,Y 511.481,Z 314.415,A -85,B 0,C 180,E1 -5476.365,E2 -5476.365} C_VEL
LIN {X 0,Y 511.158,Z 326.594,A -85,B 0,C 180,E1 -5476.837,E2 -5476.837} C_VEL
LIN {X 0,Y 510.861,Z 338.174,A -85,B 0,C 180,E1 -5477.442,E2 -5477.442} C_VEL
LIN {X 0,Y 510.562,Z 349.206,A -85,B 0,C 180,E1 -5478.184,E2 -5478.184} C_VEL
LIN {X 0,Y 510.24,Z 359.888,A -85,B 0,C 180,E1 -5479.082,E2 -5479.082} C_VEL
LIN {X 0,Y 509.891,Z 369.513,A -85,B 0,C 180,E1 -5480.079,E2 -5480.079} C_VEL
LIN {X 0,Y 509.649,Z 377.406,A -85,B 0,C 180,E1 -5481.075,E2 -5481.075} C_VEL
LIN {X 0,Y 509.459,Z 385.118,A -85,B 0,C 180,E1 -5482.27,E2 -5482.27} C_VEL
LIN {X 0,Y 509.288,Z 392.226,A -85,B 0,C 180,E1 -5483.661,E2 -5483.661} C_VEL
LIN {X 0,Y 509.241,Z 396.958,A -85,B 0,C 180,E1 -5484.853,E2 -5484.853} C_VEL
LIN {X 0,Y 509.245,Z 400.574,A -85,B 0,C 180,E1 -5486.043,E2 -5486.043} C_VEL
LIN {X 0,Y 509.2,Z 402.438,A -85,B 0,C 180,E1 -5486.835,E2 -5486.835} C_VEL
LIN {X 0,Y 509.19,Z 403.836,A -85,B 0,C 180,E1 -5487.627,E2 -5487.627} C_VEL
LIN {X 0,Y 509.079,Z 405.439,A -85,B 0,C 180,E1 -5489.209,E2 -5489.209} C_VEL
LIN {X 0,Y 509.075,Z 405.656,A -85,B 0,C 180,E1 -5490,E2 -5490} C_VEL
LIN {X 0,Y 509.112,Z 404.834,A -85,B 0,C 180,E1 -5491.582,E2 -5491.582} C_VEL
LIN {X 0,Y 509.19,Z 403.84,A -85,B 0,C 180,E1 -5492.373,E2 -5492.373} C_VEL
LIN {X 0,Y 509.2,Z 402.443,A -85,B 0,C 180,E1 -5493.164,E2 -5493.164} C_VEL
LIN {X 0,Y 509.202,Z 399.503,A -85,B 0,C 180,E1 -5494.353,E2 -5494.353} C_VEL
LIN {X 0,Y 509.282,Z 395.525,A -85,B 0,C 180,E1 -5495.543,E2 -5495.543} C_VEL
LIN {X 0,Y 509.365,Z 389.508,A -85,B 0,C 180,E1 -5496.914,E2 -5496.914} C_VEL
LIN {X 0,Y 509.493,Z 382.72,A -85,B 0,C 180,E1 -5498.128,E2 -5498.128} C_VEL
LIN {X 0,Y 509.732,Z 374.427,A -85,B 0,C 180,E1 -5499.323,E2 -5499.323} C_VEL
LIN {X 0,Y 509.968,Z 365.928,A -85,B 0,C 180,E1 -5500.32,E2 -5500.32} C_VEL
LIN {X 0,Y 510.348,Z 355.431,A -85,B 0,C 180,E1 -5501.316,E2 -5501.316} C_VEL
LIN {X 0,Y 510.646,Z 344.495,A -85,B 0,C 180,E1 -5502.154,E2 -5502.154} C_VEL
LIN {X 0,Y 510.988,Z 333.667,A -85,B 0,C 180,E1 -5502.813,E2 -5502.813} C_VEL
LIN {X 0,Y 511.267,Z 322,A -85,B 0,C 180,E1 -5503.362,E2 -5503.362} C_VEL
LIN {X 0,Y 511.548,Z 308.561,A -85,B 0,C 180,E1 -5503.81,E2 -5503.81} C_VEL
LIN {X 0,Y 511.845,Z 295.307,A -85,B 0,C 180,E1 -5504.08,E2 -5504.08} C_VEL
LIN {X 0,Y 512.111,Z 205.144,A -85,B 0,C 180,E1 -5505.352,E2 -5505.352} C_VEL
LIN {X 0,Y 510.234,Z 192.674,A -85,B 0,C 180,E1 -5505.603,E2 -5505.603} C_VEL
LIN {X 0,Y 510.723,Z 173.218,A -85,B 0,C 180,E1 -5508.659,E2 -5508.659} C_VEL
LIN {X 0,Y 511.269,Z 153.56,A -85,B 0,C 180,E1 -5511.786,E2 -5511.786} C_VEL
LIN {X 0,Y 511.358,Z 143.045,A -85,B 0,C 180,E1 -5513.488,E2 -5513.488} C_VEL
LIN {X 0,Y 509.831,Z 134.98,A -85,B 0,C 180,E1 -5514.894,E2 -5514.894} C_VEL
LIN {X 0,Y 509.844,Z 134.976,A -85,B 0,C 180,E1 -5517.057,E2 -5517.057} C_VEL
LIN {X 0,Y 509.849,Z 134.98,A -85,B 0,C 180,E1 -5519.751,E2 -5519.751} C_VEL
LIN {X 0,Y 509.842,Z 134.972,A -85,B 0,C 180,E1 -5522.768,E2 -5522.768} C_VEL
LIN {X 0,Y 509.817,Z 134.983,A -85,B 0,C 180,E1 -5525.577,E2 -5525.577} C_VEL
LIN {X 0,Y 509.844,Z 134.972,A -85,B 0,C 180,E1 -5528.337,E2 -5528.337} C_VEL
LIN {X 0,Y 509.826,Z 134.981,A -85,B 0,C 180,E1 -5531.427,E2 -5531.427} C_VEL
LIN {X 0,Y 509.833,Z 134.975,A -85,B 0,C 180,E1 -5534.669,E2 -5534.669} C_VEL
LIN {X 0,Y 509.785,Z 134.983,A -85,B 0,C 180,E1 -5537.505,E2 -5537.505} C_VEL
LIN {X 0,Y 509.825,Z 134.977,A -85,B 0,C 180,E1 -5540.645,E2 -5540.645} C_VEL
LIN {X 0,Y 509.8,Z 134.978,A -85,B 0,C 180,E1 -5543.645,E2 -5543.645} C_VEL
LIN {X 0,Y 509.83,Z 134.977,A -85,B 0,C 180,E1 -5546.537,E2 -5546.537} C_VEL
LIN {X 0,Y 509.819,Z 134.977,A -85,B 0,C 180,E1 -5549.332,E2 -5549.332} C_VEL
LIN {X 0,Y 509.823,Z 134.975,A -85,B 0,C 180,E1 -5552.05,E2 -5552.05} C_VEL
LIN {X 0,Y 509.792,Z 134.987,A -85,B 0,C 180,E1 -5554.699,E2 -5554.699} C_VEL
LIN {X 0,Y 509.814,Z 134.976,A -85,B 0,C 180,E1 -5557.458,E2 -5557.458} C_VEL
LIN {X 0,Y 509.879,Z 134.968,A -85,B 0,C 180,E1 -5559.843,E2 -5559.843} C_VEL
LIN {X 0,Y 509.835,Z 134.98,A -85,B 0,C 180,E1 -5562.346,E2 -5562.346} C_VEL
LIN {X 0,Y 509.873,Z 134.971,A -85,B 0,C 180,E1 -5564.818,E2 -5564.818} C_VEL
LIN {X 0,Y 509.878,Z 134.974,A -85,B 0,C 180,E1 -5568.131,E2 -5568.131} C_VEL
LIN {X 0,Y 509.861,Z 134.97,A -85,B 0,C 180,E1 -5571.279,E2 -5571.279} C_VEL
LIN {X 0,Y 509.905,Z 134.967,A -85,B 0,C 180,E1 -5573.669,E2 -5573.669} C_VEL
LIN {X 0,Y 509.872,Z 134.969,A -85,B 0,C 180,E1 -5576.839,E2 -5576.839} C_VEL
LIN {X 0,Y 509.911,Z 134.967,A -85,B 0,C 180,E1 -5578.42,E2 -5578.42} C_VEL
LIN {X 0,Y 510.023,Z 134.958,A -85,B 0,C 180,E1 -5580,E2 -5580} C_VEL
LIN {X 0,Y 510.031,Z 134.951,A -85,B 0,C 180,E1 -5582.369,E2 -5582.369} C_VEL
LIN {X 0,Y 509.93,Z 134.966,A -85,B 0,C 180,E1 -5585.536,E2 -5585.536} C_VEL
LIN {X 0,Y 509.889,Z 134.966,A -85,B 0,C 180,E1 -5588.721,E2 -5588.721} C_VEL
LIN {X 0,Y 509.894,Z 134.97,A -85,B 0,C 180,E1 -5591.932,E2 -5591.932} C_VEL
LIN {X 0,Y 509.885,Z 134.971,A -85,B 0,C 180,E1 -5595.242,E2 -5595.242} C_VEL
LIN {X 0,Y 509.826,Z 134.974,A -85,B 0,C 180,E1 -5598.485,E2 -5598.485} C_VEL
LIN {X 0,Y 509.834,Z 134.976,A -85,B 0,C 180,E1 -5601.002,E2 -5601.002} C_VEL
LIN {X 0,Y 509.808,Z 134.981,A -85,B 0,C 180,E1 -5603.565,E2 -5603.565} C_VEL
LIN {X 0,Y 509.809,Z 134.976,A -85,B 0,C 180,E1 -5606.358,E2 -5606.358} C_VEL
LIN {X 0,Y 509.827,Z 134.978,A -85,B 0,C 180,E1 -5608.847,E2 -5608.847} C_VEL
LIN {X 0,Y 509.809,Z 134.978,A -85,B 0,C 180,E1 -5611.591,E2 -5611.591} C_VEL
LIN {X 0,Y 509.83,Z 134.975,A -85,B 0,C 180,E1 -5614.415,E2 -5614.415} C_VEL
LIN {X 0,Y 509.809,Z 134.979,A -85,B 0,C 180,E1 -5617.342,E2 -5617.342} C_VEL
LIN {X 0,Y 509.807,Z 134.979,A -85,B 0,C 180,E1 -5620.385,E2 -5620.385} C_VEL
LIN {X 0,Y 509.789,Z 134.983,A -85,B 0,C 180,E1 -5623.06,E2 -5623.06} C_VEL
LIN {X 0,Y 509.817,Z 134.975,A -85,B 0,C 180,E1 -5625.794,E2 -5625.794} C_VEL
LIN {X 0,Y 509.841,Z 134.98,A -85,B 0,C 180,E1 -5628.574,E2 -5628.574} C_VEL
LIN {X 0,Y 509.845,Z 134.972,A -85,B 0,C 180,E1 -5631.788,E2 -5631.788} C_VEL
LIN {X 0,Y 509.804,Z 134.977,A -85,B 0,C 180,E1 -5633.695,E2 -5633.695} C_VEL
LIN {X 0,Y 509.143,Z 135.066,A -85,B 0,C 180,E1 -5634.355,E2 -5634.355} C_VEL
LIN {X 0,Y 506.341,Z 135.413,A -85,B 0,C 180,E1 -5635.427,E2 -5635.427} C_VEL
LIN {X 0,Y 503.957,Z 135.712,A -85,B 0,C 180,E1 -5636.291,E2 -5636.291} C_VEL
LIN {X 0,Y 502.909,Z 135.837,A -85,B 0,C 180,E1 -5636.957,E2 -5636.957} C_VEL
LIN {X 0,Y 502.81,Z 135.848,A -85,B 0,C 180,E1 -5637.183,E2 -5637.183} C_VEL
LIN {X 0,Y 502.808,Z 135.854,A -85,B 0,C 180,E1 -5640.067,E2 -5640.067} C_VEL
LIN {X 0,Y 502.821,Z 135.847,A -85,B 0,C 180,E1 -5643.45,E2 -5643.45} C_VEL
LIN {X 0,Y 502.768,Z 135.862,A -85,B 0,C 180,E1 -5646.086,E2 -5646.086} C_VEL
LIN {X 0,Y 502.784,Z 135.857,A -85,B 0,C 180,E1 -5648.69,E2 -5648.69} C_VEL
LIN {X 0,Y 502.9,Z 135.958,A -85,B 0,C 180,E1 -5649.899,E2 -5649.899} C_VEL
LIN {X 0,Y 503.629,Z 141.612,A -85,B 0,C 180,E1 -5651.069,E2 -5651.069} C_VEL
LIN {X 0,Y 503.267,Z 156.934,A -85,B 0,C 180,E1 -5654.035,E2 -5654.035} C_VEL
LIN {X 0,Y 503.266,Z 157.987,A -85,B 0,C 180,E1 -5654.234,E2 -5654.234} C_VEL
LIN {X 0,Y 505.447,Z 169.574,A -85,B 0,C 180,E1 -5654.489,E2 -5654.489} C_VEL
LIN {X 0,Y 504.941,Z 265.429,A -85,B 0,C 180,E1 -5655.877,E2 -5655.877} C_VEL
LIN {X 0,Y 504.737,Z 278.57,A -85,B 0,C 180,E1 -5656.231,E2 -5656.231} C_VEL
LIN {X 0,Y 504.429,Z 291.755,A -85,B 0,C 180,E1 -5656.761,E2 -5656.761} C_VEL
LIN {X 0,Y 504.146,Z 302.97,A -85,B 0,C 180,E1 -5657.378,E2 -5657.378} C_VEL
LIN {X 0,Y 503.839,Z 314.976,A -85,B 0,C 180,E1 -5658.229,E2 -5658.229} C_VEL
LIN {X 0,Y 503.46,Z 325.213,A -85,B 0,C 180,E1 -5659.138,E2 -5659.138} C_VEL
LIN {X 0,Y 503.094,Z 334.398,A -85,B 0,C 180,E1 -5660.147,E2 -5660.147} C_VEL
LIN {X 0,Y 502.778,Z 343.308,A -85,B 0,C 180,E1 -5661.358,E2 -5661.358} C_VEL
LIN {X 0,Y 502.528,Z 350.481,A -85,B 0,C 180,E1 -5662.568,E2 -5662.568} C_VEL
LIN {X 0,Y 502.415,Z 355.318,A -85,B 0,C 180,E1 -5663.575,E2 -5663.575} C_VEL
LIN {X 0,Y 502.201,Z 360.022,A -85,B 0,C 180,E1 -5664.781,E2 -5664.781} C_VEL
LIN {X 0,Y 502.248,Z 363.618,A -85,B 0,C 180,E1 -5665.988,E2 -5665.988} C_VEL
LIN {X 0,Y 502.182,Z 365.479,A -85,B 0,C 180,E1 -5666.791,E2 -5666.791} C_VEL
LIN {X 0,Y 502.131,Z 366.884,A -85,B 0,C 180,E1 -5667.594,E2 -5667.594} C_VEL
LIN {X 0,Y 501.999,Z 368.5,A -85,B 0,C 180,E1 -5669.198,E2 -5669.198} C_VEL
LIN {X 0,Y 501.992,Z 368.737,A -85,B 0,C 180,E1 -5670,E2 -5670} C_VEL
LIN {X 0,Y 501.999,Z 368.553,A -85,B 0,C 180,E1 -5670.803,E2 -5670.803} C_VEL
LIN {X 0,Y 502.131,Z 367.005,A -85,B 0,C 180,E1 -5672.407,E2 -5672.407} C_VEL
LIN {X 0,Y 502.182,Z 365.652,A -85,B 0,C 180,E1 -5673.209,E2 -5673.209} C_VEL
LIN {X 0,Y 502.25,Z 362.795,A -85,B 0,C 180,E1 -5674.414,E2 -5674.414} C_VEL
LIN {X 0,Y 502.305,Z 358.921,A -85,B 0,C 180,E1 -5675.621,E2 -5675.621} C_VEL
LIN {X 0,Y 502.403,Z 353.924,A -85,B 0,C 180,E1 -5676.829,E2 -5676.829} C_VEL
LIN {X 0,Y 502.641,Z 347.627,A -85,B 0,C 180,E1 -5678.038,E2 -5678.038} C_VEL
LIN {X 0,Y 502.877,Z 339.745,A -85,B 0,C 180,E1 -5679.249,E2 -5679.249} C_VEL
LIN {X 0,Y 503.22,Z 329.936,A -85,B 0,C 180,E1 -5680.461,E2 -5680.461} C_VEL
LIN {X 0,Y 503.622,Z 319.644,A -85,B 0,C 180,E1 -5681.47,E2 -5681.47} C_VEL
LIN {X 0,Y 503.97,Z 308.413,A -85,B 0,C 180,E1 -5682.353,E2 -5682.353} C_VEL
LIN {X 0,Y 504.327,Z 296.478,A -85,B 0,C 180,E1 -5683.088,E2 -5683.088} C_VEL
LIN {X 0,Y 504.636,Z 284.46,A -85,B 0,C 180,E1 -5683.644,E2 -5683.644} C_VEL
LIN {X 0,Y 504.889,Z 271.376,A -85,B 0,C 180,E1 -5684.074,E2 -5684.074} C_VEL
LIN {X 0,Y 505.068,Z 258.829,A -85,B 0,C 180,E1 -5684.325,E2 -5684.325} C_VEL
LIN {X 0,Y 505.448,Z 169.333,A -85,B 0,C 180,E1 -5685.605,E2 -5685.605} C_VEL
LIN {X 0,Y 503.28,Z 158.017,A -85,B 0,C 180,E1 -5685.85,E2 -5685.85} C_VEL
LIN {X 0,Y 503.648,Z 142.069,A -85,B 0,C 180,E1 -5688.931,E2 -5688.931} C_VEL
LIN {X 0,Y 502.883,Z 135.848,A -85,B 0,C 180,E1 -5690.236,E2 -5690.236} C_VEL
LIN {X 0,Y 502.789,Z 135.851,A -85,B 0,C 180,E1 -5693.041,E2 -5693.041} C_VEL
LIN {X 0,Y 502.788,Z 135.857,A -85,B 0,C 180,E1 -5695.678,E2 -5695.678} C_VEL
LIN {X 0,Y 502.798,Z 135.851,A -85,B 0,C 180,E1 -5698.375,E2 -5698.375} C_VEL
LIN {X 0,Y 502.795,Z 135.851,A -85,B 0,C 180,E1 -5701.143,E2 -5701.143} C_VEL
LIN {X 0,Y 502.805,Z 135.853,A -85,B 0,C 180,E1 -5703.994,E2 -5703.994} C_VEL
LIN {X 0,Y 502.765,Z 135.857,A -85,B 0,C 180,E1 -5707.175,E2 -5707.175} C_VEL
LIN {X 0,Y 502.773,Z 135.855,A -85,B 0,C 180,E1 -5710.016,E2 -5710.016} C_VEL
LIN {X 0,Y 502.804,Z 135.849,A -85,B 0,C 180,E1 -5712.199,E2 -5712.199} C_VEL
LIN {X 0,Y 502.785,Z 135.858,A -85,B 0,C 180,E1 -5715.47,E2 -5715.47} C_VEL
LIN {X 0,Y 502.794,Z 135.851,A -85,B 0,C 180,E1 -5717.86,E2 -5717.86} C_VEL
LIN {X 0,Y 502.792,Z 135.856,A -85,B 0,C 180,E1 -5721.023,E2 -5721.023} C_VEL
LIN {X 0,Y 502.768,Z 135.853,A -85,B 0,C 180,E1 -5724.17,E2 -5724.17} C_VEL
LIN {X 0,Y 502.801,Z 135.858,A -85,B 0,C 180,E1 -5726.999,E2 -5726.999} C_VEL
LIN {X 0,Y 502.807,Z 135.848,A -85,B 0,C 180,E1 -5730.066,E2 -5730.066} C_VEL
LIN {X 0,Y 502.821,Z 135.848,A -85,B 0,C 180,E1 -5733.448,E2 -5733.448} C_VEL
LIN {X 0,Y 502.764,Z 135.855,A -85,B 0,C 180,E1 -5736.085,E2 -5736.085} C_VEL
LIN {X 0,Y 502.777,Z 135.861,A -85,B 0,C 180,E1 -5738.688,E2 -5738.688} C_VEL
LIN {X 0,Y 502.803,Z 135.85,A -85,B 0,C 180,E1 -5741.247,E2 -5741.247} C_VEL
LIN {X 0,Y 502.832,Z 135.852,A -85,B 0,C 180,E1 -5744.665,E2 -5744.665} C_VEL
LIN {X 0,Y 502.874,Z 135.843,A -85,B 0,C 180,E1 -5748.039,E2 -5748.039} C_VEL
LIN {X 0,Y 502.844,Z 135.844,A -85,B 0,C 180,E1 -5751.156,E2 -5751.156} C_VEL
LIN {X 0,Y 502.862,Z 135.842,A -85,B 0,C 180,E1 -5753.58,E2 -5753.58} C_VEL
LIN {X 0,Y 502.827,Z 135.847,A -85,B 0,C 180,E1 -5756.795,E2 -5756.795} C_VEL
LIN {X 0,Y 502.888,Z 135.843,A -85,B 0,C 180,E1 -5758.398,E2 -5758.398} C_VEL
LIN {X 0,Y 502.998,Z 135.832,A -85,B 0,C 180,E1 -5760,E2 -5760} C_VEL
LIN {X 0,Y 503.003,Z 135.827,A -85,B 0,C 180,E1 -5762.402,E2 -5762.402} C_VEL
LIN {X 0,Y 502.886,Z 135.843,A -85,B 0,C 180,E1 -5765.614,E2 -5765.614} C_VEL
LIN {X 0,Y 502.841,Z 135.85,A -85,B 0,C 180,E1 -5768.034,E2 -5768.034} C_VEL
LIN {X 0,Y 502.831,Z 135.848,A -85,B 0,C 180,E1 -5771.284,E2 -5771.284} C_VEL
LIN {X 0,Y 502.793,Z 135.85,A -85,B 0,C 180,E1 -5774.572,E2 -5774.572} C_VEL
LIN {X 0,Y 502.779,Z 135.856,A -85,B 0,C 180,E1 -5777.91,E2 -5777.91} C_VEL
LIN {X 0,Y 502.799,Z 135.849,A -85,B 0,C 180,E1 -5780.528,E2 -5780.528} C_VEL
LIN {X 0,Y 502.775,Z 135.856,A -85,B 0,C 180,E1 -5783.041,E2 -5783.041} C_VEL
LIN {X 0,Y 502.772,Z 135.857,A -85,B 0,C 180,E1 -5785.679,E2 -5785.679} C_VEL
LIN {X 0,Y 502.756,Z 135.855,A -85,B 0,C 180,E1 -5788.378,E2 -5788.378} C_VEL
LIN {X 0,Y 502.767,Z 135.858,A -85,B 0,C 180,E1 -5791.494,E2 -5791.494} C_VEL
LIN {X 0,Y 502.783,Z 135.852,A -85,B 0,C 180,E1 -5794.441,E2 -5794.441} C_VEL
LIN {X 0,Y 502.76,Z 135.861,A -85,B 0,C 180,E1 -5797.176,E2 -5797.176} C_VEL
LIN {X 0,Y 502.769,Z 135.853,A -85,B 0,C 180,E1 -5800.017,E2 -5800.017} C_VEL
LIN {X 0,Y 502.745,Z 135.859,A -85,B 0,C 180,E1 -5803.234,E2 -5803.234} C_VEL
LIN {X 0,Y 502.777,Z 135.852,A -85,B 0,C 180,E1 -5805.66,E2 -5805.66} C_VEL
LIN {X 0,Y 502.764,Z 135.858,A -85,B 0,C 180,E1 -5809.013,E2 -5809.013} C_VEL
LIN {X 0,Y 502.789,Z 135.852,A -85,B 0,C 180,E1 -5812.046,E2 -5812.046} C_VEL
LIN {X 0,Y 502.792,Z 135.852,A -85,B 0,C 180,E1 -5815.034,E2 -5815.034} C_VEL
LIN {X 0,Y 502.783,Z 135.854,A -85,B 0,C 180,E1 -5817.915,E2 -5817.915} C_VEL
LIN {X 0,Y 502.806,Z 135.854,A -85,B 0,C 180,E1 -5820.711,E2 -5820.711} C_VEL
LIN {X 0,Y 502.776,Z 135.857,A -85,B 0,C 180,E1 -5823.46,E2 -5823.46} C_VEL
LIN {X 0,Y 502.809,Z 135.988,A -85,B 0,C 180,E1 -5824.96,E2 -5824.96} C_VEL
LIN {X 0,Y 504.493,Z 145.144,A -85,B 0,C 180,E1 -5826.561,E2 -5826.561} C_VEL
LIN {X 0,Y 504.143,Z 159.952,A -85,B 0,C 180,E1 -5828.977,E2 -5828.977} C_VEL
LIN {X 0,Y 503.559,Z 179.496,A -85,B 0,C 180,E1 -5832.119,E2 -5832.119} C_VEL
LIN {X 0,Y 503.222,Z 192.712,A -85,B 0,C 180,E1 -5834.194,E2 -5834.194} C_VEL
LIN {X 0,Y 505.298,Z 206.926,A -85,B 0,C 180,E1 -5834.465,E2 -5834.465} C_VEL
LIN {X 0,Y 504.876,Z 300.868,A -85,B 0,C 180,E1 -5835.823,E2 -5835.823} C_VEL
LIN {X 0,Y 504.584,Z 314.158,A -85,B 0,C 180,E1 -5836.175,E2 -5836.175} C_VEL
LIN {X 0,Y 504.244,Z 326.336,A -85,B 0,C 180,E1 -5836.653,E2 -5836.653} C_VEL
LIN {X 0,Y 503.899,Z 338.473,A -85,B 0,C 180,E1 -5837.3,E2 -5837.3} C_VEL
LIN {X 0,Y 503.562,Z 348.945,A -85,B 0,C 180,E1 -5838.018,E2 -5838.018} C_VEL
LIN {X 0,Y 503.22,Z 359.627,A -85,B 0,C 180,E1 -5838.928,E2 -5838.928} C_VEL
LIN {X 0,Y 502.839,Z 369.252,A -85,B 0,C 180,E1 -5839.938,E2 -5839.938} C_VEL
LIN {X 0,Y 502.605,Z 377.146,A -85,B 0,C 180,E1 -5840.949,E2 -5840.949} C_VEL
LIN {X 0,Y 502.38,Z 384.857,A -85,B 0,C 180,E1 -5842.16,E2 -5842.16} C_VEL
LIN {X 0,Y 502.236,Z 391.558,A -85,B 0,C 180,E1 -5843.482,E2 -5843.482} C_VEL
LIN {X 0,Y 502.171,Z 396.699,A -85,B 0,C 180,E1 -5844.78,E2 -5844.78} C_VEL
LIN {X 0,Y 502.138,Z 400.314,A -85,B 0,C 180,E1 -5845.987,E2 -5845.987} C_VEL
LIN {X 0,Y 502.12,Z 402.179,A -85,B 0,C 180,E1 -5846.79,E2 -5846.79} C_VEL
LIN {X 0,Y 502.092,Z 403.577,A -85,B 0,C 180,E1 -5847.593,E2 -5847.593} C_VEL
LIN {X 0,Y 501.995,Z 405.181,A -85,B 0,C 180,E1 -5849.197,E2 -5849.197} C_VEL
LIN {X 0,Y 501.989,Z 405.398,A -85,B 0,C 180,E1 -5850,E2 -5850} C_VEL
LIN {X 0,Y 502.036,Z 404.575,A -85,B 0,C 180,E1 -5851.604,E2 -5851.604} C_VEL
LIN {X 0,Y 502.092,Z 403.581,A -85,B 0,C 180,E1 -5852.406,E2 -5852.406} C_VEL
LIN {X 0,Y 502.12,Z 402.184,A -85,B 0,C 180,E1 -5853.209,E2 -5853.209} C_VEL
LIN {X 0,Y 502.1,Z 399.243,A -85,B 0,C 180,E1 -5854.415,E2 -5854.415} C_VEL
LIN {X 0,Y 502.197,Z 395.266,A -85,B 0,C 180,E1 -5855.621,E2 -5855.621} C_VEL
LIN {X 0,Y 502.29,Z 389.248,A -85,B 0,C 180,E1 -5857.012,E2 -5857.012} C_VEL
LIN {X 0,Y 502.447,Z 382.46,A -85,B 0,C 180,E1 -5858.242,E2 -5858.242} C_VEL
LIN {X 0,Y 502.705,Z 374.167,A -85,B 0,C 180,E1 -5859.454,E2 -5859.454} C_VEL
LIN {X 0,Y 502.957,Z 365.668,A -85,B 0,C 180,E1 -5860.465,E2 -5860.465} C_VEL
LIN {X 0,Y 503.363,Z 355.171,A -85,B 0,C 180,E1 -5861.476,E2 -5861.476} C_VEL
LIN {X 0,Y 503.69,Z 344.235,A -85,B 0,C 180,E1 -5862.324,E2 -5862.324} C_VEL
LIN {X 0,Y 504.03,Z 333.405,A -85,B 0,C 180,E1 -5862.993,E2 -5862.993} C_VEL
LIN {X 0,Y 504.332,Z 321.738,A -85,B 0,C 180,E1 -5863.549,E2 -5863.549} C_VEL
LIN {X 0,Y 504.665,Z 308.299,A -85,B 0,C 180,E1 -5864.002,E2 -5864.002} C_VEL
LIN {X 0,Y 504.962,Z 295.042,A -85,B 0,C 180,E1 -5864.276,E2 -5864.276} C_VEL
LIN {X 0,Y 505.201,Z 205.559,A -85,B 0,C 180,E1 -5865.558,E2 -5865.558} C_VEL
LIN {X 0,Y 503.213,Z 192.454,A -85,B 0,C 180,E1 -5865.819,E2 -5865.819} C_VEL
LIN {X 0,Y 503.734,Z 174.269,A -85,B 0,C 180,E1 -5868.716,E2 -5868.716} C_VEL
LIN {X 0,Y 504.313,Z 154.617,A -85,B 0,C 180,E1 -5871.886,E2 -5871.886} C_VEL
LIN {X 0,Y 504.489,Z 145.161,A -85,B 0,C 180,E1 -5873.435,E2 -5873.435} C_VEL
LIN {X 0,Y 502.786,Z 135.858,A -85,B 0,C 180,E1 -5875.068,E2 -5875.068} C_VEL
LIN {X 0,Y 502.788,Z 135.857,A -85,B 0,C 180,E1 -5877.469,E2 -5877.469} C_VEL
LIN {X 0,Y 502.8,Z 135.853,A -85,B 0,C 180,E1 -5880.211,E2 -5880.211} C_VEL
LIN {X 0,Y 502.799,Z 135.851,A -85,B 0,C 180,E1 -5883.033,E2 -5883.033} C_VEL
LIN {X 0,Y 502.763,Z 135.856,A -85,B 0,C 180,E1 -5885.951,E2 -5885.951} C_VEL
LIN {X 0,Y 502.791,Z 135.853,A -85,B 0,C 180,E1 -5888.976,E2 -5888.976} C_VEL
LIN {X 0,Y 502.766,Z 135.854,A -85,B 0,C 180,E1 -5892.194,E2 -5892.194} C_VEL
LIN {X 0,Y 502.779,Z 135.857,A -85,B 0,C 180,E1 -5895.469,E2 -5895.469} C_VEL
LIN {X 0,Y 502.759,Z 135.855,A -85,B 0,C 180,E1 -5897.857,E2 -5897.857} C_VEL
LIN {X 0,Y 502.785,Z 135.859,A -85,B 0,C 180,E1 -5901.022,E2 -5901.022} C_VEL
LIN {X 0,Y 502.762,Z 135.854,A -85,B 0,C 180,E1 -5904.169,E2 -5904.169} C_VEL
LIN {X 0,Y 502.794,Z 135.857,A -85,B 0,C 180,E1 -5906.998,E2 -5906.998} C_VEL
LIN {X 0,Y 502.8,Z 135.85,A -85,B 0,C 180,E1 -5910.066,E2 -5910.066} C_VEL
LIN {X 0,Y 502.774,Z 135.853,A -85,B 0,C 180,E1 -5913.429,E2 -5913.429} C_VEL
LIN {X 0,Y 502.754,Z 135.857,A -85,B 0,C 180,E1 -5916.084,E2 -5916.084} C_VEL
LIN {X 0,Y 502.82,Z 135.847,A -85,B 0,C 180,E1 -5919.463,E2 -5919.463} C_VEL
LIN {X 0,Y 502.773,Z 135.856,A -85,B 0,C 180,E1 -5922.09,E2 -5922.09} C_VEL
LIN {X 0,Y 502.814,Z 135.847,A -85,B 0,C 180,E1 -5925.428,E2 -5925.428} C_VEL
LIN {X 0,Y 502.826,Z 135.849,A -85,B 0,C 180,E1 -5928.716,E2 -5928.716} C_VEL
LIN {X 0,Y 502.835,Z 135.85,A -85,B 0,C 180,E1 -5931.966,E2 -5931.966} C_VEL
LIN {X 0,Y 502.881,Z 135.844,A -85,B 0,C 180,E1 -5934.386,E2 -5934.386} C_VEL
LIN {X 0,Y 502.997,Z 135.827,A -85,B 0,C 180,E1 -5937.598,E2 -5937.598} C_VEL
LIN {X 0,Y 502.992,Z 135.834,A -85,B 0,C 180,E1 -5940,E2 -5940} C_VEL
LIN {X 0,Y 502.998,Z 135.827,A -85,B 0,C 180,E1 -5942.402,E2 -5942.402} C_VEL
LIN {X 0,Y 502.886,Z 135.844,A -85,B 0,C 180,E1 -5945.614,E2 -5945.614} C_VEL
LIN {X 0,Y 502.86,Z 135.846,A -85,B 0,C 180,E1 -5948.034,E2 -5948.034} C_VEL
LIN {X 0,Y 502.865,Z 135.845,A -85,B 0,C 180,E1 -5951.284,E2 -5951.284} C_VEL
LIN {X 0,Y 502.815,Z 135.847,A -85,B 0,C 180,E1 -5954.572,E2 -5954.572} C_VEL
LIN {X 0,Y 502.799,Z 135.85,A -85,B 0,C 180,E1 -5958.109,E2 -5958.109} C_VEL
LIN {X 0,Y 502.82,Z 135.847,A -85,B 0,C 180,E1 -5960.537,E2 -5960.537} C_VEL
LIN {X 0,Y 502.776,Z 135.857,A -85,B 0,C 180,E1 -5963.041,E2 -5963.041} C_VEL
LIN {X 0,Y 502.768,Z 135.856,A -85,B 0,C 180,E1 -5965.68,E2 -5965.68} C_VEL
LIN {X 0,Y 502.764,Z 135.854,A -85,B 0,C 180,E1 -5968.378,E2 -5968.378} C_VEL
LIN {X 0,Y 502.784,Z 135.859,A -85,B 0,C 180,E1 -5971.144,E2 -5971.144} C_VEL
LIN {X 0,Y 502.781,Z 135.852,A -85,B 0,C 180,E1 -5973.996,E2 -5973.996} C_VEL
LIN {X 0,Y 502.77,Z 135.858,A -85,B 0,C 180,E1 -5977.178,E2 -5977.178} C_VEL
LIN {X 0,Y 502.764,Z 135.854,A -85,B 0,C 180,E1 -5980.018,E2 -5980.018} C_VEL
LIN {X 0,Y 502.744,Z 135.859,A -85,B 0,C 180,E1 -5983.235,E2 -5983.235} C_VEL
LIN {X 0,Y 502.774,Z 135.852,A -85,B 0,C 180,E1 -5985.661,E2 -5985.661} C_VEL
LIN {X 0,Y 502.791,Z 135.854,A -85,B 0,C 180,E1 -5988.933,E2 -5988.933} C_VEL
LIN {X 0,Y 502.786,Z 135.853,A -85,B 0,C 180,E1 -5992.047,E2 -5992.047} C_VEL
LIN {X 0,Y 502.794,Z 135.851,A -85,B 0,C 180,E1 -5995.035,E2 -5995.035} C_VEL
LIN {X 0,Y 502.81,Z 135.848,A -85,B 0,C 180,E1 -5997.183,E2 -5997.183} C_VEL
LIN {X 0,Y 502.107,Z 135.939,A -85,B 0,C 180,E1 -5997.852,E2 -5997.852} C_VEL
LIN {X 0,Y 499.245,Z 136.297,A -85,B 0,C 180,E1 -5998.937,E2 -5998.937} C_VEL
LIN {X 0,Y 496.845,Z 136.597,A -85,B 0,C 180,E1 -5999.812,E2 -5999.812} C_VEL
LIN {X 0,Y 495.812,Z 136.725,A -85,B 0,C 180,E1 -6000.488,E2 -6000.488} C_VEL
LIN {X 0,Y 495.725,Z 136.733,A -85,B 0,C 180,E1 -6000.717,E2 -6000.717} C_VEL
LIN {X 0,Y 495.742,Z 136.733,A -85,B 0,C 180,E1 -6003.93,E2 -6003.93} C_VEL
LIN {X 0,Y 495.758,Z 136.727,A -85,B 0,C 180,E1 -6007.141,E2 -6007.141} C_VEL
LIN {X 0,Y 495.857,Z 136.74,A -85,B 0,C 180,E1 -6009.741,E2 -6009.741} C_VEL
LIN {X 0,Y 496.664,Z 142.81,A -85,B 0,C 180,E1 -6011.007,E2 -6011.007} C_VEL
LIN {X 0,Y 496.285,Z 158.282,A -85,B 0,C 180,E1 -6014.019,E2 -6014.019} C_VEL
LIN {X 0,Y 498.64,Z 170.8,A -85,B 0,C 180,E1 -6014.285,E2 -6014.285} C_VEL
LIN {X 0,Y 498.088,Z 265.708,A -85,B 0,C 180,E1 -6015.679,E2 -6015.679} C_VEL
LIN {X 0,Y 497.87,Z 278.842,A -85,B 0,C 180,E1 -6016.038,E2 -6016.038} C_VEL
LIN {X 0,Y 497.563,Z 290.914,A -85,B 0,C 180,E1 -6016.523,E2 -6016.523} C_VEL
LIN {X 0,Y 497.27,Z 302.691,A -85,B 0,C 180,E1 -6017.165,E2 -6017.165} C_VEL
LIN {X 0,Y 496.952,Z 313.955,A -85,B 0,C 180,E1 -6017.96,E2 -6017.96} C_VEL
LIN {X 0,Y 496.496,Z 324.419,A -85,B 0,C 180,E1 -6018.881,E2 -6018.881} C_VEL
LIN {X 0,Y 496.174,Z 332.964,A -85,B 0,C 180,E1 -6019.802,E2 -6019.802} C_VEL
LIN {X 0,Y 495.899,Z 340.832,A -85,B 0,C 180,E1 -6020.826,E2 -6020.826} C_VEL
LIN {X 0,Y 495.56,Z 348.527,A -85,B 0,C 180,E1 -6022.053,E2 -6022.053} C_VEL
LIN {X 0,Y 495.349,Z 355.58,A -85,B 0,C 180,E1 -6023.483,E2 -6023.483} C_VEL
LIN {X 0,Y 495.142,Z 360.283,A -85,B 0,C 180,E1 -6024.707,E2 -6024.707} C_VEL
LIN {X 0,Y 495.186,Z 363.878,A -85,B 0,C 180,E1 -6025.931,E2 -6025.931} C_VEL
LIN {X 0,Y 495.103,Z 365.74,A -85,B 0,C 180,E1 -6026.745,E2 -6026.745} C_VEL
LIN {X 0,Y 495.065,Z 367.143,A -85,B 0,C 180,E1 -6027.56,E2 -6027.56} C_VEL
LIN {X 0,Y 494.919,Z 368.759,A -85,B 0,C 180,E1 -6029.187,E2 -6029.187} C_VEL
LIN {X 0,Y 494.909,Z 368.995,A -85,B 0,C 180,E1 -6030,E2 -6030} C_VEL
LIN {X 0,Y 494.919,Z 368.811,A -85,B 0,C 180,E1 -6030.814,E2 -6030.814} C_VEL
LIN {X 0,Y 495.066,Z 367.262,A -85,B 0,C 180,E1 -6032.441,E2 -6032.441} C_VEL
LIN {X 0,Y 495.103,Z 365.91,A -85,B 0,C 180,E1 -6033.255,E2 -6033.255} C_VEL
LIN {X 0,Y 495.178,Z 363.053,A -85,B 0,C 180,E1 -6034.477,E2 -6034.477} C_VEL
LIN {X 0,Y 495.257,Z 359.178,A -85,B 0,C 180,E1 -6035.701,E2 -6035.701} C_VEL
LIN {X 0,Y 495.364,Z 354.18,A -85,B 0,C 180,E1 -6036.926,E2 -6036.926} C_VEL
LIN {X 0,Y 495.599,Z 347.883,A -85,B 0,C 180,E1 -6038.153,E2 -6038.153} C_VEL
LIN {X 0,Y 495.858,Z 340.001,A -85,B 0,C 180,E1 -6039.381,E2 -6039.381} C_VEL
LIN {X 0,Y 496.204,Z 331.961,A -85,B 0,C 180,E1 -6040.404,E2 -6040.404} C_VEL
LIN {X 0,Y 496.599,Z 322.149,A -85,B 0,C 180,E1 -6041.428,E2 -6041.428} C_VEL
LIN {X 0,Y 496.921,Z 312.497,A -85,B 0,C 180,E1 -6042.248,E2 -6042.248} C_VEL
LIN {X 0,Y 497.289,Z 301.68,A -85,B 0,C 180,E1 -6042.988,E2 -6042.988} C_VEL
LIN {X 0,Y 497.609,Z 289.485,A -85,B 0,C 180,E1 -6043.632,E2 -6043.632} C_VEL
LIN {X 0,Y 497.937,Z 276.138,A -85,B 0,C 180,E1 -6044.144,E2 -6044.144} C_VEL
LIN {X 0,Y 498.153,Z 263.639,A -85,B 0,C 180,E1 -6044.45,E2 -6044.45} C_VEL
LIN {X 0,Y 498.561,Z 170.054,A -85,B 0,C 180,E1 -6045.819,E2 -6045.819} C_VEL
LIN {X 0,Y 496.284,Z 158.256,A -85,B 0,C 180,E1 -6046.078,E2 -6046.078} C_VEL
LIN {X 0,Y 496.675,Z 142.199,A -85,B 0,C 180,E1 -6049.208,E2 -6049.208} C_VEL
LIN {X 0,Y 495.823,Z 136.727,A -85,B 0,C 180,E1 -6050.38,E2 -6050.38} C_VEL
LIN {X 0,Y 495.742,Z 136.73,A -85,B 0,C 180,E1 -6053.388,E2 -6053.388} C_VEL
LIN {X 0,Y 495.776,Z 136.724,A -85,B 0,C 180,E1 -6056.737,E2 -6056.737} C_VEL
LIN {X 0,Y 495.764,Z 136.734,A -85,B 0,C 180,E1 -6059.746,E2 -6059.746} C_VEL
LIN {X 0,Y 495.769,Z 136.725,A -85,B 0,C 180,E1 -6062.594,E2 -6062.594} C_VEL
LIN {X 0,Y 495.746,Z 136.735,A -85,B 0,C 180,E1 -6065.538,E2 -6065.538} C_VEL
LIN {X 0,Y 495.758,Z 136.727,A -85,B 0,C 180,E1 -6068.767,E2 -6068.767} C_VEL
LIN {X 0,Y 495.745,Z 136.732,A -85,B 0,C 180,E1 -6071.782,E2 -6071.782} C_VEL
LIN {X 0,Y 495.737,Z 136.735,A -85,B 0,C 180,E1 -6075.141,E2 -6075.141} C_VEL
LIN {X 0,Y 495.744,Z 136.728,A -85,B 0,C 180,E1 -6078.217,E2 -6078.217} C_VEL
LIN {X 0,Y 495.744,Z 136.733,A -85,B 0,C 180,E1 -6081.408,E2 -6081.408} C_VEL
LIN {X 0,Y 495.741,Z 136.73,A -85,B 0,C 180,E1 -6084.461,E2 -6084.461} C_VEL
LIN {X 0,Y 495.748,Z 136.731,A -85,B 0,C 180,E1 -6087.404,E2 -6087.404} C_VEL
LIN {X 0,Y 495.754,Z 136.728,A -85,B 0,C 180,E1 -6090.253,E2 -6090.253} C_VEL
LIN {X 0,Y 495.771,Z 136.728,A -85,B 0,C 180,E1 -6093.262,E2 -6093.262} C_VEL
LIN {X 0,Y 495.736,Z 136.736,A -85,B 0,C 180,E1 -6096.612,E2 -6096.612} C_VEL
LIN {X 0,Y 495.776,Z 136.725,A -85,B 0,C 180,E1 -6099.324,E2 -6099.324} C_VEL
LIN {X 0,Y 495.776,Z 136.725,A -85,B 0,C 180,E1 -6101.828,E2 -6101.828} C_VEL
LIN {X 0,Y 495.772,Z 136.725,A -85,B 0,C 180,E1 -6105.217,E2 -6105.217} C_VEL
LIN {X 0,Y 495.847,Z 136.722,A -85,B 0,C 180,E1 -6108.555,E2 -6108.555} C_VEL
LIN {X 0,Y 495.809,Z 136.723,A -85,B 0,C 180,E1 -6111.851,E2 -6111.851} C_VEL
LIN {X 0,Y 495.846,Z 136.723,A -85,B 0,C 180,E1 -6114.306,E2 -6114.306} C_VEL
LIN {X 0,Y 495.971,Z 136.701,A -85,B 0,C 180,E1 -6117.564,E2 -6117.564} C_VEL
LIN {X 0,Y 495.967,Z 136.708,A -85,B 0,C 180,E1 -6120,E2 -6120} C_VEL
LIN {X 0,Y 495.97,Z 136.703,A -85,B 0,C 180,E1 -6122.436,E2 -6122.436} C_VEL
LIN {X 0,Y 495.844,Z 136.721,A -85,B 0,C 180,E1 -6125.694,E2 -6125.694} C_VEL
LIN {X 0,Y 495.805,Z 136.725,A -85,B 0,C 180,E1 -6128.149,E2 -6128.149} C_VEL
LIN {X 0,Y 495.809,Z 136.724,A -85,B 0,C 180,E1 -6131.446,E2 -6131.446} C_VEL
LIN {X 0,Y 495.741,Z 136.729,A -85,B 0,C 180,E1 -6134.784,E2 -6134.784} C_VEL
LIN {X 0,Y 495.744,Z 136.729,A -85,B 0,C 180,E1 -6138.226,E2 -6138.226} C_VEL
LIN {X 0,Y 495.742,Z 136.729,A -85,B 0,C 180,E1 -6140.758,E2 -6140.758} C_VEL
LIN {X 0,Y 495.726,Z 136.739,A -85,B 0,C 180,E1 -6143.388,E2 -6143.388} C_VEL
LIN {X 0,Y 495.735,Z 136.731,A -85,B 0,C 180,E1 -6146.729,E2 -6146.729} C_VEL
LIN {X 0,Y 495.692,Z 136.737,A -85,B 0,C 180,E1 -6149.751,E2 -6149.751} C_VEL
LIN {X 0,Y 495.745,Z 136.73,A -85,B 0,C 180,E1 -6152.596,E2 -6152.596} C_VEL
LIN {X 0,Y 495.737,Z 136.732,A -85,B 0,C 180,E1 -6155.539,E2 -6155.539} C_VEL
LIN {X 0,Y 495.755,Z 136.732,A -85,B 0,C 180,E1 -6158.767,E2 -6158.767} C_VEL
LIN {X 0,Y 495.722,Z 136.731,A -85,B 0,C 180,E1 -6161.785,E2 -6161.785} C_VEL
LIN {X 0,Y 495.736,Z 136.733,A -85,B 0,C 180,E1 -6165.141,E2 -6165.141} C_VEL
LIN {X 0,Y 495.723,Z 136.733,A -85,B 0,C 180,E1 -6168.216,E2 -6168.216} C_VEL
LIN {X 0,Y 495.746,Z 136.728,A -85,B 0,C 180,E1 -6171.408,E2 -6171.408} C_VEL
LIN {X 0,Y 495.743,Z 136.736,A -85,B 0,C 180,E1 -6174.462,E2 -6174.462} C_VEL
LIN {X 0,Y 495.752,Z 136.727,A -85,B 0,C 180,E1 -6177.405,E2 -6177.405} C_VEL
LIN {X 0,Y 495.759,Z 136.734,A -85,B 0,C 180,E1 -6180.253,E2 -6180.253} C_VEL
LIN {X 0,Y 495.741,Z 136.733,A -85,B 0,C 180,E1 -6183.27,E2 -6183.27} C_VEL
LIN {X 0,Y 495.776,Z 136.882,A -85,B 0,C 180,E1 -6184.776,E2 -6184.776} C_VEL
LIN {X 0,Y 497.454,Z 145.432,A -85,B 0,C 180,E1 -6186.3,E2 -6186.3} C_VEL
LIN {X 0,Y 497.489,Z 151.743,A -85,B 0,C 180,E1 -6187.359,E2 -6187.359} C_VEL
LIN {X 0,Y 496.917,Z 168.778,A -85,B 0,C 180,E1 -6190.157,E2 -6190.157} C_VEL
LIN {X 0,Y 496.36,Z 187.074,A -85,B 0,C 180,E1 -6193.126,E2 -6193.126} C_VEL
LIN {X 0,Y 496.218,Z 192.375,A -85,B 0,C 180,E1 -6193.964,E2 -6193.964} C_VEL
LIN {X 0,Y 498.477,Z 208.122,A -85,B 0,C 180,E1 -6194.268,E2 -6194.268} C_VEL
LIN {X 0,Y 497.988,Z 300.615,A -85,B 0,C 180,E1 -6195.623,E2 -6195.623} C_VEL
LIN {X 0,Y 497.669,Z 313.903,A -85,B 0,C 180,E1 -6195.979,E2 -6195.979} C_VEL
LIN {X 0,Y 497.332,Z 326.08,A -85,B 0,C 180,E1 -6196.464,E2 -6196.464} C_VEL
LIN {X 0,Y 496.994,Z 336.759,A -85,B 0,C 180,E1 -6197.032,E2 -6197.032} C_VEL
LIN {X 0,Y 496.613,Z 347.369,A -85,B 0,C 180,E1 -6197.744,E2 -6197.744} C_VEL
LIN {X 0,Y 496.235,Z 358.293,A -85,B 0,C 180,E1 -6198.667,E2 -6198.667} C_VEL
LIN {X 0,Y 495.86,Z 367.201,A -85,B 0,C 180,E1 -6199.589,E2 -6199.589} C_VEL
LIN {X 0,Y 495.562,Z 376.886,A -85,B 0,C 180,E1 -6200.819,E2 -6200.819} C_VEL
LIN {X 0,Y 495.318,Z 384.597,A -85,B 0,C 180,E1 -6202.048,E2 -6202.048} C_VEL
LIN {X 0,Y 495.172,Z 389.881,A -85,B 0,C 180,E1 -6203.071,E2 -6203.071} C_VEL
LIN {X 0,Y 495.112,Z 395.004,A -85,B 0,C 180,E1 -6204.297,E2 -6204.297} C_VEL
LIN {X 0,Y 495.006,Z 398.98,A -85,B 0,C 180,E1 -6205.521,E2 -6205.521} C_VEL
LIN {X 0,Y 495.042,Z 401.92,A -85,B 0,C 180,E1 -6206.744,E2 -6206.744} C_VEL
LIN {X 0,Y 494.998,Z 403.317,A -85,B 0,C 180,E1 -6207.558,E2 -6207.558} C_VEL
LIN {X 0,Y 494.962,Z 404.314,A -85,B 0,C 180,E1 -6208.372,E2 -6208.372} C_VEL
LIN {X 0,Y 494.906,Z 405.139,A -85,B 0,C 180,E1 -6210,E2 -6210} C_VEL
LIN {X 0,Y 494.962,Z 404.317,A -85,B 0,C 180,E1 -6211.627,E2 -6211.627} C_VEL
LIN {X 0,Y 494.998,Z 403.322,A -85,B 0,C 180,E1 -6212.441,E2 -6212.441} C_VEL
LIN {X 0,Y 495.041,Z 401.925,A -85,B 0,C 180,E1 -6213.255,E2 -6213.255} C_VEL
LIN {X 0,Y 495.005,Z 398.983,A -85,B 0,C 180,E1 -6214.478,E2 -6214.478} C_VEL
LIN {X 0,Y 495.113,Z 395.006,A -85,B 0,C 180,E1 -6215.702,E2 -6215.702} C_VEL
LIN {X 0,Y 495.239,Z 388.887,A -85,B 0,C 180,E1 -6217.132,E2 -6217.132} C_VEL
LIN {X 0,Y 495.404,Z 382.2,A -85,B 0,C 180,E1 -6218.36,E2 -6218.36} C_VEL
LIN {X 0,Y 495.67,Z 373.906,A -85,B 0,C 180,E1 -6219.59,E2 -6219.59} C_VEL
LIN {X 0,Y 495.96,Z 365.407,A -85,B 0,C 180,E1 -6220.615,E2 -6220.615} C_VEL
LIN {X 0,Y 496.375,Z 354.909,A -85,B 0,C 180,E1 -6221.639,E2 -6221.639} C_VEL
LIN {X 0,Y 496.752,Z 343.155,A -85,B 0,C 180,E1 -6222.559,E2 -6222.559} C_VEL
LIN {X 0,Y 497.15,Z 331.219,A -85,B 0,C 180,E1 -6223.28,E2 -6223.28} C_VEL
LIN {X 0,Y 497.511,Z 318.869,A -85,B 0,C 180,E1 -6223.842,E2 -6223.842} C_VEL
LIN {X 0,Y 497.867,Z 306.204,A -85,B 0,C 180,E1 -6224.249,E2 -6224.249} C_VEL
LIN {X 0,Y 498.074,Z 292.998,A -85,B 0,C 180,E1 -6224.504,E2 -6224.504} C_VEL
LIN {X 0,Y 498.357,Z 206.359,A -85,B 0,C 180,E1 -6225.761,E2 -6225.761} C_VEL
LIN {X 0,Y 496.24,Z 192.148,A -85,B 0,C 180,E1 -6226.054,E2 -6226.054} C_VEL
LIN {X 0,Y 496.736,Z 174.009,A -85,B 0,C 180,E1 -6228.99,E2 -6228.99} C_VEL
LIN {X 0,Y 497.397,Z 154.36,A -85,B 0,C 180,E1 -6232.207,E2 -6232.207} C_VEL
LIN {X 0,Y 497.553,Z 146.484,A -85,B 0,C 180,E1 -6233.517,E2 -6233.517} C_VEL
LIN {X 0,Y 495.747,Z 136.736,A -85,B 0,C 180,E1 -6235.281,E2 -6235.281} C_VEL
LIN {X 0,Y 495.722,Z 136.737,A -85,B 0,C 180,E1 -6237.894,E2 -6237.894} C_VEL
LIN {X 0,Y 495.744,Z 136.73,A -85,B 0,C 180,E1 -6240.687,E2 -6240.687} C_VEL
LIN {X 0,Y 495.737,Z 136.738,A -85,B 0,C 180,E1 -6243.565,E2 -6243.565} C_VEL
LIN {X 0,Y 495.712,Z 136.732,A -85,B 0,C 180,E1 -6246.544,E2 -6246.544} C_VEL
LIN {X 0,Y 495.741,Z 136.733,A -85,B 0,C 180,E1 -6249.638,E2 -6249.638} C_VEL
LIN {X 0,Y 495.708,Z 136.733,A -85,B 0,C 180,E1 -6252.503,E2 -6252.503} C_VEL
LIN {X 0,Y 495.731,Z 136.737,A -85,B 0,C 180,E1 -6255.14,E2 -6255.14} C_VEL
LIN {X 0,Y 495.716,Z 136.732,A -85,B 0,C 180,E1 -6258.215,E2 -6258.215} C_VEL
LIN {X 0,Y 495.738,Z 136.733,A -85,B 0,C 180,E1 -6261.407,E2 -6261.407} C_VEL
LIN {X 0,Y 495.734,Z 136.732,A -85,B 0,C 180,E1 -6264.461,E2 -6264.461} C_VEL
LIN {X 0,Y 495.742,Z 136.73,A -85,B 0,C 180,E1 -6267.404,E2 -6267.404} C_VEL
LIN {X 0,Y 495.747,Z 136.73,A -85,B 0,C 180,E1 -6270.252,E2 -6270.252} C_VEL
LIN {X 0,Y 495.73,Z 136.732,A -85,B 0,C 180,E1 -6273.27,E2 -6273.27} C_VEL
LIN {X 0,Y 495.727,Z 136.739,A -85,B 0,C 180,E1 -6276.612,E2 -6276.612} C_VEL
LIN {X 0,Y 495.769,Z 136.725,A -85,B 0,C 180,E1 -6279.324,E2 -6279.324} C_VEL
LIN {X 0,Y 495.75,Z 136.729,A -85,B 0,C 180,E1 -6281.827,E2 -6281.827} C_VEL
LIN {X 0,Y 495.765,Z 136.726,A -85,B 0,C 180,E1 -6285.216,E2 -6285.216} C_VEL
LIN {X 0,Y 495.811,Z 136.725,A -85,B 0,C 180,E1 -6288.554,E2 -6288.554} C_VEL
LIN {X 0,Y 495.799,Z 136.725,A -85,B 0,C 180,E1 -6291.851,E2 -6291.851} C_VEL
LIN {X 0,Y 495.839,Z 136.722,A -85,B 0,C 180,E1 -6294.306,E2 -6294.306} C_VEL
LIN {X 0,Y 495.964,Z 136.703,A -85,B 0,C 180,E1 -6297.564,E2 -6297.564} C_VEL
LIN {X 0,Y 495.961,Z 136.71,A -85,B 0,C 180,E1 -6300,E2 -6300} C_VEL
LIN {X 0,Y 495.965,Z 136.703,A -85,B 0,C 180,E1 -6302.436,E2 -6302.436} C_VEL
LIN {X 0,Y 495.844,Z 136.723,A -85,B 0,C 180,E1 -6305.694,E2 -6305.694} C_VEL
LIN {X 0,Y 495.819,Z 136.722,A -85,B 0,C 180,E1 -6308.149,E2 -6308.149} C_VEL
LIN {X 0,Y 495.84,Z 136.722,A -85,B 0,C 180,E1 -6311.446,E2 -6311.446} C_VEL
LIN {X 0,Y 495.766,Z 136.726,A -85,B 0,C 180,E1 -6314.784,E2 -6314.784} C_VEL
LIN {X 0,Y 495.762,Z 136.726,A -85,B 0,C 180,E1 -6318.235,E2 -6318.235} C_VEL
LIN {X 0,Y 495.765,Z 136.727,A -85,B 0,C 180,E1 -6320.757,E2 -6320.757} C_VEL
LIN {X 0,Y 495.729,Z 136.738,A -85,B 0,C 180,E1 -6323.388,E2 -6323.388} C_VEL
LIN {X 0,Y 495.73,Z 136.732,A -85,B 0,C 180,E1 -6326.73,E2 -6326.73} C_VEL
LIN {X 0,Y 495.748,Z 136.729,A -85,B 0,C 180,E1 -6329.748,E2 -6329.748} C_VEL
LIN {X 0,Y 495.744,Z 136.731,A -85,B 0,C 180,E1 -6332.596,E2 -6332.596} C_VEL
LIN {X 0,Y 495.739,Z 136.73,A -85,B 0,C 180,E1 -6335.539,E2 -6335.539} C_VEL
LIN {X 0,Y 495.751,Z 136.734,A -85,B 0,C 180,E1 -6338.768,E2 -6338.768} C_VEL
LIN {X 0,Y 495.719,Z 136.731,A -85,B 0,C 180,E1 -6341.785,E2 -6341.785} C_VEL
LIN {X 0,Y 495.732,Z 136.733,A -85,B 0,C 180,E1 -6345.142,E2 -6345.142} C_VEL
LIN {X 0,Y 495.745,Z 136.731,A -85,B 0,C 180,E1 -6348.219,E2 -6348.219} C_VEL
LIN {X 0,Y 495.743,Z 136.728,A -85,B 0,C 180,E1 -6351.409,E2 -6351.409} C_VEL
LIN {X 0,Y 495.742,Z 136.737,A -85,B 0,C 180,E1 -6354.463,E2 -6354.463} C_VEL
LIN {X 0,Y 495.765,Z 136.726,A -85,B 0,C 180,E1 -6357.407,E2 -6357.407} C_VEL
LIN {X 0,Y 495.756,Z 136.735,A -85,B 0,C 180,E1 -6360.254,E2 -6360.254} C_VEL
LIN {X 0,Y 495.725,Z 136.733,A -85,B 0,C 180,E1 -6360.717,E2 -6360.717} C_VEL
LIN {X 0,Y 495.047,Z 136.816,A -85,B 0,C 180,E1 -6361.395,E2 -6361.395} C_VEL
LIN {X 0,Y 492.184,Z 137.176,A -85,B 0,C 180,E1 -6362.498,E2 -6362.498} C_VEL
LIN {X 0,Y 489.781,Z 137.473,A -85,B 0,C 180,E1 -6363.386,E2 -6363.386} C_VEL
LIN {X 0,Y 488.767,Z 137.604,A -85,B 0,C 180,E1 -6364.072,E2 -6364.072} C_VEL
LIN {X 0,Y 488.694,Z 137.61,A -85,B 0,C 180,E1 -6364.304,E2 -6364.304} C_VEL
LIN {X 0,Y 488.721,Z 137.603,A -85,B 0,C 180,E1 -6367.154,E2 -6367.154} C_VEL
LIN {X 0,Y 488.788,Z 137.636,A -85,B 0,C 180,E1 -6369.596,E2 -6369.596} C_VEL
LIN {X 0,Y 489.689,Z 142.961,A -85,B 0,C 180,E1 -6370.726,E2 -6370.726} C_VEL
LIN {X 0,Y 489.322,Z 158.26,A -85,B 0,C 180,E1 -6373.736,E2 -6373.736} C_VEL
LIN {X 0,Y 489.325,Z 158.55,A -85,B 0,C 180,E1 -6373.789,E2 -6373.789} C_VEL
LIN {X 0,Y 491.824,Z 171.713,A -85,B 0,C 180,E1 -6374.071,E2 -6374.071} C_VEL
LIN {X 0,Y 491.222,Z 265.987,A -85,B 0,C 180,E1 -6375.474,E2 -6375.474} C_VEL
LIN {X 0,Y 491.006,Z 279.114,A -85,B 0,C 180,E1 -6375.838,E2 -6375.838} C_VEL
LIN {X 0,Y 490.64,Z 292.292,A -85,B 0,C 180,E1 -6376.382,E2 -6376.382} C_VEL
LIN {X 0,Y 490.351,Z 303.498,A -85,B 0,C 180,E1 -6377.016,E2 -6377.016} C_VEL
LIN {X 0,Y 490.025,Z 314.219,A -85,B 0,C 180,E1 -6377.788,E2 -6377.788} C_VEL
LIN {X 0,Y 489.537,Z 324.682,A -85,B 0,C 180,E1 -6378.72,E2 -6378.72} C_VEL
LIN {X 0,Y 489.198,Z 333.227,A -85,B 0,C 180,E1 -6379.655,E2 -6379.655} C_VEL
LIN {X 0,Y 488.889,Z 341.094,A -85,B 0,C 180,E1 -6380.694,E2 -6380.694} C_VEL
LIN {X 0,Y 488.537,Z 348.788,A -85,B 0,C 180,E1 -6381.938,E2 -6381.938} C_VEL
LIN {X 0,Y 488.31,Z 355.841,A -85,B 0,C 180,E1 -6383.389,E2 -6383.389} C_VEL
LIN {X 0,Y 488.087,Z 360.543,A -85,B 0,C 180,E1 -6384.63,E2 -6384.63} C_VEL
LIN {X 0,Y 488.106,Z 364.138,A -85,B 0,C 180,E1 -6385.872,E2 -6385.872} C_VEL
LIN {X 0,Y 488.028,Z 365.999,A -85,B 0,C 180,E1 -6386.698,E2 -6386.698} C_VEL
LIN {X 0,Y 487.972,Z 367.403,A -85,B 0,C 180,E1 -6387.524,E2 -6387.524} C_VEL
LIN {X 0,Y 487.841,Z 369.018,A -85,B 0,C 180,E1 -6389.175,E2 -6389.175} C_VEL
LIN {X 0,Y 487.829,Z 369.254,A -85,B 0,C 180,E1 -6390,E2 -6390} C_VEL
LIN {X 0,Y 487.841,Z 369.069,A -85,B 0,C 180,E1 -6390.826,E2 -6390.826} C_VEL
LIN {X 0,Y 487.973,Z 367.521,A -85,B 0,C 180,E1 -6392.477,E2 -6392.477} C_VEL
LIN {X 0,Y 488.028,Z 366.168,A -85,B 0,C 180,E1 -6393.303,E2 -6393.303} C_VEL
LIN {X 0,Y 488.089,Z 363.311,A -85,B 0,C 180,E1 -6394.543,E2 -6394.543} C_VEL
LIN {X 0,Y 488.21,Z 359.435,A -85,B 0,C 180,E1 -6395.784,E2 -6395.784} C_VEL
LIN {X 0,Y 488.324,Z 354.437,A -85,B 0,C 180,E1 -6397.027,E2 -6397.027} C_VEL
LIN {X 0,Y 488.561,Z 348.14,A -85,B 0,C 180,E1 -6398.271,E2 -6398.271} C_VEL
LIN {X 0,Y 488.856,Z 340.256,A -85,B 0,C 180,E1 -6399.517,E2 -6399.517} C_VEL
LIN {X 0,Y 489.223,Z 332.217,A -85,B 0,C 180,E1 -6400.554,E2 -6400.554} C_VEL
LIN {X 0,Y 489.648,Z 322.404,A -85,B 0,C 180,E1 -6401.592,E2 -6401.592} C_VEL
LIN {X 0,Y 489.992,Z 312.751,A -85,B 0,C 180,E1 -6402.424,E2 -6402.424} C_VEL
LIN {X 0,Y 490.381,Z 302.014,A -85,B 0,C 180,E1 -6403.169,E2 -6403.169} C_VEL
LIN {X 0,Y 490.728,Z 289.734,A -85,B 0,C 180,E1 -6403.827,E2 -6403.827} C_VEL
LIN {X 0,Y 491.056,Z 277.154,A -85,B 0,C 180,E1 -6404.32,E2 -6404.32} C_VEL
LIN {X 0,Y 491.293,Z 265.297,A -85,B 0,C 180,E1 -6404.63,E2 -6404.63} C_VEL
LIN {X 0,Y 491.691,Z 170.661,A -85,B 0,C 180,E1 -6406.04,E2 -6406.04} C_VEL
LIN {X 0,Y 489.326,Z 158.514,A -85,B 0,C 180,E1 -6406.307,E2 -6406.307} C_VEL
LIN {X 0,Y 489.72,Z 143.414,A -85,B 0,C 180,E1 -6409.273,E2 -6409.273} C_VEL
LIN {X 0,Y 488.776,Z 137.604,A -85,B 0,C 180,E1 -6410.536,E2 -6410.536} C_VEL
LIN {X 0,Y 488.673,Z 137.614,A -85,B 0,C 180,E1 -6413.747,E2 -6413.747} C_VEL
LIN {X 0,Y 488.726,Z 137.602,A -85,B 0,C 180,E1 -6416.928,E2 -6416.928} C_VEL
LIN {X 0,Y 488.724,Z 137.606,A -85,B 0,C 180,E1 -6420.219,E2 -6420.219} C_VEL
LIN {X 0,Y 488.736,Z 137.607,A -85,B 0,C 180,E1 -6423.484,E2 -6423.484} C_VEL
LIN {X 0,Y 488.674,Z 137.609,A -85,B 0,C 180,E1 -6426.353,E2 -6426.353} C_VEL
LIN {X 0,Y 488.694,Z 137.611,A -85,B 0,C 180,E1 -6429.255,E2 -6429.255} C_VEL
LIN {X 0,Y 488.689,Z 137.607,A -85,B 0,C 180,E1 -6432.526,E2 -6432.526} C_VEL
LIN {X 0,Y 488.701,Z 137.612,A -85,B 0,C 180,E1 -6435.197,E2 -6435.197} C_VEL
LIN {X 0,Y 488.679,Z 137.609,A -85,B 0,C 180,E1 -6438.581,E2 -6438.581} C_VEL
LIN {X 0,Y 488.673,Z 137.61,A -85,B 0,C 180,E1 -6441.799,E2 -6441.799} C_VEL
LIN {X 0,Y 488.716,Z 137.612,A -85,B 0,C 180,E1 -6445.053,E2 -6445.053} C_VEL
LIN {X 0,Y 488.696,Z 137.606,A -85,B 0,C 180,E1 -6448.047,E2 -6448.047} C_VEL
LIN {X 0,Y 488.698,Z 137.612,A -85,B 0,C 180,E1 -6450.728,E2 -6450.728} C_VEL
LIN {X 0,Y 488.709,Z 137.605,A -85,B 0,C 180,E1 -6453.525,E2 -6453.525} C_VEL
LIN {X 0,Y 488.667,Z 137.612,A -85,B 0,C 180,E1 -6456.253,E2 -6456.253} C_VEL
LIN {X 0,Y 488.744,Z 137.602,A -85,B 0,C 180,E1 -6459.176,E2 -6459.176} C_VEL
LIN {X 0,Y 488.744,Z 137.6,A -85,B 0,C 180,E1 -6461.632,E2 -6461.632} C_VEL
LIN {X 0,Y 488.743,Z 137.603,A -85,B 0,C 180,E1 -6464.999,E2 -6464.999} C_VEL
LIN {X 0,Y 488.802,Z 137.601,A -85,B 0,C 180,E1 -6468.387,E2 -6468.387} C_VEL
LIN {X 0,Y 488.757,Z 137.6,A -85,B 0,C 180,E1 -6471.733,E2 -6471.733} C_VEL
LIN {X 0,Y 488.806,Z 137.601,A -85,B 0,C 180,E1 -6474.224,E2 -6474.224} C_VEL
LIN {X 0,Y 488.937,Z 137.577,A -85,B 0,C 180,E1 -6477.528,E2 -6477.528} C_VEL
LIN {X 0,Y 488.936,Z 137.584,A -85,B 0,C 180,E1 -6480,E2 -6480} C_VEL
LIN {X 0,Y 488.936,Z 137.579,A -85,B 0,C 180,E1 -6482.471,E2 -6482.471} C_VEL
LIN {X 0,Y 488.804,Z 137.599,A -85,B 0,C 180,E1 -6485.776,E2 -6485.776} C_VEL
LIN {X 0,Y 488.749,Z 137.602,A -85,B 0,C 180,E1 -6488.268,E2 -6488.268} C_VEL
LIN {X 0,Y 488.77,Z 137.604,A -85,B 0,C 180,E1 -6491.613,E2 -6491.613} C_VEL
LIN {X 0,Y 488.71,Z 137.605,A -85,B 0,C 180,E1 -6495.002,E2 -6495.002} C_VEL
LIN {X 0,Y 488.702,Z 137.606,A -85,B 0,C 180,E1 -6498.444,E2 -6498.444} C_VEL
LIN {X 0,Y 488.686,Z 137.611,A -85,B 0,C 180,E1 -6501.072,E2 -6501.072} C_VEL
LIN {X 0,Y 488.656,Z 137.615,A -85,B 0,C 180,E1 -6503.747,E2 -6503.747} C_VEL
LIN {X 0,Y 488.678,Z 137.609,A -85,B 0,C 180,E1 -6506.477,E2 -6506.477} C_VEL
LIN {X 0,Y 488.656,Z 137.619,A -85,B 0,C 180,E1 -6509.275,E2 -6509.275} C_VEL
LIN {X 0,Y 488.687,Z 137.607,A -85,B 0,C 180,E1 -6512.148,E2 -6512.148} C_VEL
LIN {X 0,Y 488.708,Z 137.613,A -85,B 0,C 180,E1 -6515.116,E2 -6515.116} C_VEL
LIN {X 0,Y 488.672,Z 137.61,A -85,B 0,C 180,E1 -6518.201,E2 -6518.201} C_VEL
LIN {X 0,Y 488.692,Z 137.608,A -85,B 0,C 180,E1 -6520.341,E2 -6520.341} C_VEL
LIN {X 0,Y 488.672,Z 137.609,A -85,B 0,C 180,E1 -6523.656,E2 -6523.656} C_VEL
LIN {X 0,Y 488.672,Z 137.612,A -85,B 0,C 180,E1 -6526.344,E2 -6526.344} C_VEL
LIN {X 0,Y 488.703,Z 137.605,A -85,B 0,C 180,E1 -6529.674,E2 -6529.674} C_VEL
LIN {X 0,Y 488.67,Z 137.614,A -85,B 0,C 180,E1 -6532.84,E2 -6532.84} C_VEL
LIN {X 0,Y 488.718,Z 137.605,A -85,B 0,C 180,E1 -6535.886,E2 -6535.886} C_VEL
LIN {X 0,Y 488.69,Z 137.612,A -85,B 0,C 180,E1 -6538.82,E2 -6538.82} C_VEL
LIN {X 0,Y 488.697,Z 137.61,A -85,B 0,C 180,E1 -6541.668,E2 -6541.668} C_VEL
LIN {X 0,Y 488.723,Z 137.742,A -85,B 0,C 180,E1 -6544.58,E2 -6544.58} C_VEL
LIN {X 0,Y 490.632,Z 148.154,A -85,B 0,C 180,E1 -6546.457,E2 -6546.457} C_VEL
LIN {X 0,Y 490.12,Z 164.596,A -85,B 0,C 180,E1 -6549.213,E2 -6549.213} C_VEL
LIN {X 0,Y 489.494,Z 182.899,A -85,B 0,C 180,E1 -6552.236,E2 -6552.236} C_VEL
LIN {X 0,Y 489.242,Z 192.101,A -85,B 0,C 180,E1 -6553.728,E2 -6553.728} C_VEL
LIN {X 0,Y 491.649,Z 209.281,A -85,B 0,C 180,E1 -6554.065,E2 -6554.065} C_VEL
LIN {X 0,Y 491.107,Z 300.365,A -85,B 0,C 180,E1 -6555.417,E2 -6555.417} C_VEL
LIN {X 0,Y 490.798,Z 313.65,A -85,B 0,C 180,E1 -6555.778,E2 -6555.778} C_VEL
LIN {X 0,Y 490.441,Z 325.825,A -85,B 0,C 180,E1 -6556.27,E2 -6556.27} C_VEL
LIN {X 0,Y 490.058,Z 336.422,A -85,B 0,C 180,E1 -6556.84,E2 -6556.84} C_VEL
LIN {X 0,Y 489.646,Z 347.111,A -85,B 0,C 180,E1 -6557.567,E2 -6557.567} C_VEL
LIN {X 0,Y 489.261,Z 358.035,A -85,B 0,C 180,E1 -6558.503,E2 -6558.503} C_VEL
LIN {X 0,Y 488.847,Z 366.942,A -85,B 0,C 180,E1 -6559.438,E2 -6559.438} C_VEL
LIN {X 0,Y 488.51,Z 376.626,A -85,B 0,C 180,E1 -6560.685,E2 -6560.685} C_VEL
LIN {X 0,Y 488.244,Z 384.337,A -85,B 0,C 180,E1 -6561.932,E2 -6561.932} C_VEL
LIN {X 0,Y 488.089,Z 389.621,A -85,B 0,C 180,E1 -6562.97,E2 -6562.97} C_VEL
LIN {X 0,Y 488.007,Z 394.744,A -85,B 0,C 180,E1 -6564.214,E2 -6564.214} C_VEL
LIN {X 0,Y 487.918,Z 398.72,A -85,B 0,C 180,E1 -6565.456,E2 -6565.456} C_VEL
LIN {X 0,Y 487.964,Z 401.661,A -85,B 0,C 180,E1 -6566.697,E2 -6566.697} C_VEL
LIN {X 0,Y 487.891,Z 404.056,A -85,B 0,C 180,E1 -6568.349,E2 -6568.349} C_VEL
LIN {X 0,Y 487.827,Z 404.881,A -85,B 0,C 180,E1 -6570,E2 -6570} C_VEL
LIN {X 0,Y 487.891,Z 404.059,A -85,B 0,C 180,E1 -6571.65,E2 -6571.65} C_VEL
LIN {X 0,Y 487.964,Z 401.666,A -85,B 0,C 180,E1 -6573.302,E2 -6573.302} C_VEL
LIN {X 0,Y 487.918,Z 398.723,A -85,B 0,C 180,E1 -6574.543,E2 -6574.543} C_VEL
LIN {X 0,Y 488.009,Z 394.744,A -85,B 0,C 180,E1 -6575.785,E2 -6575.785} C_VEL
LIN {X 0,Y 488.173,Z 388.626,A -85,B 0,C 180,E1 -6577.236,E2 -6577.236} C_VEL
LIN {X 0,Y 488.341,Z 381.938,A -85,B 0,C 180,E1 -6578.482,E2 -6578.482} C_VEL
LIN {X 0,Y 488.637,Z 373.644,A -85,B 0,C 180,E1 -6579.729,E2 -6579.729} C_VEL
LIN {X 0,Y 488.972,Z 365.146,A -85,B 0,C 180,E1 -6580.768,E2 -6580.768} C_VEL
LIN {X 0,Y 489.38,Z 354.646,A -85,B 0,C 180,E1 -6581.808,E2 -6581.808} C_VEL
LIN {X 0,Y 489.802,Z 343.057,A -85,B 0,C 180,E1 -6582.728,E2 -6582.728} C_VEL
LIN {X 0,Y 490.225,Z 330.956,A -85,B 0,C 180,E1 -6583.471,E2 -6583.471} C_VEL
LIN {X 0,Y 490.615,Z 318.605,A -85,B 0,C 180,E1 -6584.041,E2 -6584.041} C_VEL
LIN {X 0,Y 490.987,Z 305.938,A -85,B 0,C 180,E1 -6584.453,E2 -6584.453} C_VEL
LIN {X 0,Y 491.195,Z 292.725,A -85,B 0,C 180,E1 -6584.712,E2 -6584.712} C_VEL
LIN {X 0,Y 491.588,Z 207.568,A -85,B 0,C 180,E1 -6585.962,E2 -6585.962} C_VEL
LIN {X 0,Y 489.221,Z 191.947,A -85,B 0,C 180,E1 -6586.281,E2 -6586.281} C_VEL
LIN {X 0,Y 489.774,Z 173.749,A -85,B 0,C 180,E1 -6589.27,E2 -6589.27} C_VEL
LIN {X 0,Y 490.455,Z 155.415,A -85,B 0,C 180,E1 -6592.316,E2 -6592.316} C_VEL
LIN {X 0,Y 490.602,Z 147.537,A -85,B 0,C 180,E1 -6593.647,E2 -6593.647} C_VEL
LIN {X 0,Y 488.725,Z 137.611,A -85,B 0,C 180,E1 -6595.453,E2 -6595.453} C_VEL
LIN {X 0,Y 488.683,Z 137.611,A -85,B 0,C 180,E1 -6598.685,E2 -6598.685} C_VEL
LIN {X 0,Y 488.686,Z 137.613,A -85,B 0,C 180,E1 -6601.179,E2 -6601.179} C_VEL
LIN {X 0,Y 488.714,Z 137.605,A -85,B 0,C 180,E1 -6604.113,E2 -6604.113} C_VEL
LIN {X 0,Y 488.666,Z 137.614,A -85,B 0,C 180,E1 -6607.159,E2 -6607.159} C_VEL
LIN {X 0,Y 488.688,Z 137.607,A -85,B 0,C 180,E1 -6610.34,E2 -6610.34} C_VEL
LIN {X 0,Y 488.671,Z 137.613,A -85,B 0,C 180,E1 -6613.655,E2 -6613.655} C_VEL
LIN {X 0,Y 488.667,Z 137.61,A -85,B 0,C 180,E1 -6616.343,E2 -6616.343} C_VEL
LIN {X 0,Y 488.696,Z 137.608,A -85,B 0,C 180,E1 -6619.673,E2 -6619.673} C_VEL
LIN {X 0,Y 488.662,Z 137.617,A -85,B 0,C 180,E1 -6622.839,E2 -6622.839} C_VEL
LIN {X 0,Y 488.709,Z 137.605,A -85,B 0,C 180,E1 -6625.885,E2 -6625.885} C_VEL
LIN {X 0,Y 488.677,Z 137.617,A -85,B 0,C 180,E1 -6628.819,E2 -6628.819} C_VEL
LIN {X 0,Y 488.685,Z 137.608,A -85,B 0,C 180,E1 -6631.667,E2 -6631.667} C_VEL
LIN {X 0,Y 488.689,Z 137.611,A -85,B 0,C 180,E1 -6634.959,E2 -6634.959} C_VEL
LIN {X 0,Y 488.679,Z 137.61,A -85,B 0,C 180,E1 -6638.042,E2 -6638.042} C_VEL
LIN {X 0,Y 488.716,Z 137.61,A -85,B 0,C 180,E1 -6640.686,E2 -6640.686} C_VEL
LIN {X 0,Y 488.659,Z 137.611,A -85,B 0,C 180,E1 -6643.283,E2 -6643.283} C_VEL
LIN {X 0,Y 488.71,Z 137.607,A -85,B 0,C 180,E1 -6645.849,E2 -6645.849} C_VEL
LIN {X 0,Y 488.773,Z 137.604,A -85,B 0,C 180,E1 -6648.387,E2 -6648.387} C_VEL
LIN {X 0,Y 488.745,Z 137.603,A -85,B 0,C 180,E1 -6651.732,E2 -6651.732} C_VEL
LIN {X 0,Y 488.799,Z 137.601,A -85,B 0,C 180,E1 -6654.224,E2 -6654.224} C_VEL
LIN {X 0,Y 488.93,Z 137.579,A -85,B 0,C 180,E1 -6657.529,E2 -6657.529} C_VEL
LIN {X 0,Y 488.93,Z 137.585,A -85,B 0,C 180,E1 -6660,E2 -6660} C_VEL
LIN {X 0,Y 488.931,Z 137.579,A -85,B 0,C 180,E1 -6662.472,E2 -6662.472} C_VEL
LIN {X 0,Y 488.804,Z 137.601,A -85,B 0,C 180,E1 -6665.776,E2 -6665.776} C_VEL
LIN {X 0,Y 488.768,Z 137.599,A -85,B 0,C 180,E1 -6668.267,E2 -6668.267} C_VEL
LIN {X 0,Y 488.795,Z 137.602,A -85,B 0,C 180,E1 -6671.613,E2 -6671.613} C_VEL
LIN {X 0,Y 488.736,Z 137.603,A -85,B 0,C 180,E1 -6675.001,E2 -6675.001} C_VEL
LIN {X 0,Y 488.734,Z 137.601,A -85,B 0,C 180,E1 -6678.443,E2 -6678.443} C_VEL
LIN {X 0,Y 488.697,Z 137.61,A -85,B 0,C 180,E1 -6681.071,E2 -6681.071} C_VEL
LIN {X 0,Y 488.659,Z 137.614,A -85,B 0,C 180,E1 -6683.747,E2 -6683.747} C_VEL
LIN {X 0,Y 488.689,Z 137.611,A -85,B 0,C 180,E1 -6686.922,E2 -6686.922} C_VEL
LIN {X 0,Y 488.71,Z 137.605,A -85,B 0,C 180,E1 -6690.22,E2 -6690.22} C_VEL
LIN {X 0,Y 488.703,Z 137.608,A -85,B 0,C 180,E1 -6693.481,E2 -6693.481} C_VEL
LIN {X 0,Y 488.675,Z 137.61,A -85,B 0,C 180,E1 -6696.355,E2 -6696.355} C_VEL
LIN {X 0,Y 488.687,Z 137.611,A -85,B 0,C 180,E1 -6699.256,E2 -6699.256} C_VEL
LIN {X 0,Y 488.66,Z 137.616,A -85,B 0,C 180,E1 -6702.529,E2 -6702.529} C_VEL
LIN {X 0,Y 488.696,Z 137.608,A -85,B 0,C 180,E1 -6705.198,E2 -6705.198} C_VEL
LIN {X 0,Y 488.688,Z 137.615,A -85,B 0,C 180,E1 -6708.584,E2 -6708.584} C_VEL
LIN {X 0,Y 488.696,Z 137.609,A -85,B 0,C 180,E1 -6710.949,E2 -6710.949} C_VEL
LIN {X 0,Y 488.666,Z 137.611,A -85,B 0,C 180,E1 -6713.868,E2 -6713.868} C_VEL
LIN {X 0,Y 488.736,Z 137.603,A -85,B 0,C 180,E1 -6716.878,E2 -6716.878} C_VEL
LIN {X 0,Y 488.716,Z 137.606,A -85,B 0,C 180,E1 -6719.781,E2 -6719.781} C_VEL
LIN {X 0,Y 488.721,Z 137.603,A -85,B 0,C 180,E1 -6723.074,E2 -6723.074} C_VEL
LIN {X 0,Y 488.694,Z 137.61,A -85,B 0,C 180,E1 -6724.304,E2 -6724.304} C_VEL
LIN {X 0,Y 488.052,Z 137.694,A -85,B 0,C 180,E1 -6724.992,E2 -6724.992} C_VEL
LIN {X 0,Y 485.205,Z 138.05,A -85,B 0,C 180,E1 -6726.109,E2 -6726.109} C_VEL
LIN {X 0,Y 482.776,Z 138.35,A -85,B 0,C 180,E1 -6727.009,E2 -6727.009} C_VEL
LIN {X 0,Y 481.725,Z 138.479,A -85,B 0,C 180,E1 -6727.705,E2 -6727.705} C_VEL
LIN {X 0,Y 481.636,Z 138.489,A -85,B 0,C 180,E1 -6727.94,E2 -6727.94} C_VEL
LIN {X 0,Y 481.75,Z 138.537,A -85,B 0,C 180,E1 -6729.447,E2 -6729.447} C_VEL
LIN {X 0,Y 482.717,Z 145.248,A -85,B 0,C 180,E1 -6730.873,E2 -6730.873} C_VEL
LIN {X 0,Y 482.367,Z 158.844,A -85,B 0,C 180,E1 -6733.548,E2 -6733.548} C_VEL
LIN {X 0,Y 485.047,Z 172.984,A -85,B 0,C 180,E1 -6733.858,E2 -6733.858} C_VEL
LIN {X 0,Y 484.369,Z 266.265,A -85,B 0,C 180,E1 -6735.264,E2 -6735.264} C_VEL
LIN {X 0,Y 484.126,Z 279.386,A -85,B 0,C 180,E1 -6735.633,E2 -6735.633} C_VEL
LIN {X 0,Y 483.754,Z 292.56,A -85,B 0,C 180,E1 -6736.185,E2 -6736.185} C_VEL
LIN {X 0,Y 483.419,Z 304.157,A -85,B 0,C 180,E1 -6736.854,E2 -6736.854} C_VEL
LIN {X 0,Y 483.056,Z 315.769,A -85,B 0,C 180,E1 -6737.715,E2 -6737.715} C_VEL
LIN {X 0,Y 482.566,Z 326.005,A -85,B 0,C 180,E1 -6738.662,E2 -6738.662} C_VEL
LIN {X 0,Y 482.126,Z 335.186,A -85,B 0,C 180,E1 -6739.714,E2 -6739.714} C_VEL
LIN {X 0,Y 481.722,Z 344.095,A -85,B 0,C 180,E1 -6740.977,E2 -6740.977} C_VEL
LIN {X 0,Y 481.396,Z 351.267,A -85,B 0,C 180,E1 -6742.239,E2 -6742.239} C_VEL
LIN {X 0,Y 481.238,Z 357.084,A -85,B 0,C 180,E1 -6743.525,E2 -6743.525} C_VEL
LIN {X 0,Y 480.95,Z 362.119,A -85,B 0,C 180,E1 -6744.971,E2 -6744.971} C_VEL
LIN {X 0,Y 481.028,Z 364.398,A -85,B 0,C 180,E1 -6745.811,E2 -6745.811} C_VEL
LIN {X 0,Y 480.956,Z 366.259,A -85,B 0,C 180,E1 -6746.65,E2 -6746.65} C_VEL
LIN {X 0,Y 480.884,Z 367.663,A -85,B 0,C 180,E1 -6747.488,E2 -6747.488} C_VEL
LIN {X 0,Y 480.767,Z 369.276,A -85,B 0,C 180,E1 -6749.163,E2 -6749.163} C_VEL
LIN {X 0,Y 480.753,Z 369.512,A -85,B 0,C 180,E1 -6750,E2 -6750} C_VEL
LIN {X 0,Y 480.767,Z 369.327,A -85,B 0,C 180,E1 -6750.838,E2 -6750.838} C_VEL
LIN {X 0,Y 480.884,Z 367.779,A -85,B 0,C 180,E1 -6752.513,E2 -6752.513} C_VEL
LIN {X 0,Y 480.956,Z 366.426,A -85,B 0,C 180,E1 -6753.351,E2 -6753.351} C_VEL
LIN {X 0,Y 481.006,Z 363.569,A -85,B 0,C 180,E1 -6754.61,E2 -6754.61} C_VEL
LIN {X 0,Y 481.164,Z 359.692,A -85,B 0,C 180,E1 -6755.869,E2 -6755.869} C_VEL
LIN {X 0,Y 481.278,Z 354.692,A -85,B 0,C 180,E1 -6757.13,E2 -6757.13} C_VEL
LIN {X 0,Y 481.539,Z 348.397,A -85,B 0,C 180,E1 -6758.393,E2 -6758.393} C_VEL
LIN {X 0,Y 481.863,Z 340.512,A -85,B 0,C 180,E1 -6759.656,E2 -6759.656} C_VEL
LIN {X 0,Y 482.217,Z 332.473,A -85,B 0,C 180,E1 -6760.709,E2 -6760.709} C_VEL
LIN {X 0,Y 482.699,Z 322.658,A -85,B 0,C 180,E1 -6761.762,E2 -6761.762} C_VEL
LIN {X 0,Y 483.13,Z 311.65,A -85,B 0,C 180,E1 -6762.709,E2 -6762.709} C_VEL
LIN {X 0,Y 483.541,Z 300.805,A -85,B 0,C 180,E1 -6763.448,E2 -6763.448} C_VEL
LIN {X 0,Y 483.906,Z 288.856,A -85,B 0,C 180,E1 -6764.08,E2 -6764.08} C_VEL
LIN {X 0,Y 484.237,Z 275.76,A -85,B 0,C 180,E1 -6764.579,E2 -6764.579} C_VEL
LIN {X 0,Y 484.484,Z 262.601,A -85,B 0,C 180,E1 -6764.894,E2 -6764.894} C_VEL
LIN {X 0,Y 484.977,Z 172.111,A -85,B 0,C 180,E1 -6766.25,E2 -6766.25} C_VEL
LIN {X 0,Y 482.387,Z 158.747,A -85,B 0,C 180,E1 -6766.549,E2 -6766.549} C_VEL
LIN {X 0,Y 482.767,Z 144.732,A -85,B 0,C 180,E1 -6769.323,E2 -6769.323} C_VEL
LIN {X 0,Y 481.735,Z 138.48,A -85,B 0,C 180,E1 -6770.674,E2 -6770.674} C_VEL
LIN {X 0,Y 481.651,Z 138.491,A -85,B 0,C 180,E1 -6774.115,E2 -6774.115} C_VEL
LIN {X 0,Y 481.696,Z 138.479,A -85,B 0,C 180,E1 -6777.126,E2 -6777.126} C_VEL
LIN {X 0,Y 481.674,Z 138.489,A -85,B 0,C 180,E1 -6779.741,E2 -6779.741} C_VEL
LIN {X 0,Y 481.674,Z 138.481,A -85,B 0,C 180,E1 -6782.674,E2 -6782.674} C_VEL
LIN {X 0,Y 481.662,Z 138.485,A -85,B 0,C 180,E1 -6785.204,E2 -6785.204} C_VEL
LIN {X 0,Y 481.666,Z 138.483,A -85,B 0,C 180,E1 -6788.859,E2 -6788.859} C_VEL
LIN {X 0,Y 481.641,Z 138.486,A -85,B 0,C 180,E1 -6792.161,E2 -6792.161} C_VEL
LIN {X 0,Y 481.654,Z 138.489,A -85,B 0,C 180,E1 -6795.542,E2 -6795.542} C_VEL
LIN {X 0,Y 481.633,Z 138.49,A -85,B 0,C 180,E1 -6798.956,E2 -6798.956} C_VEL
LIN {X 0,Y 481.647,Z 138.485,A -85,B 0,C 180,E1 -6801.994,E2 -6801.994} C_VEL
LIN {X 0,Y 481.68,Z 138.485,A -85,B 0,C 180,E1 -6805.317,E2 -6805.317} C_VEL
LIN {X 0,Y 481.637,Z 138.487,A -85,B 0,C 180,E1 -6808.311,E2 -6808.311} C_VEL
LIN {X 0,Y 481.658,Z 138.487,A -85,B 0,C 180,E1 -6811.216,E2 -6811.216} C_VEL
LIN {X 0,Y 481.658,Z 138.483,A -85,B 0,C 180,E1 -6814.04,E2 -6814.04} C_VEL
LIN {X 0,Y 481.672,Z 138.489,A -85,B 0,C 180,E1 -6816.812,E2 -6816.812} C_VEL
LIN {X 0,Y 481.69,Z 138.479,A -85,B 0,C 180,E1 -6819.502,E2 -6819.502} C_VEL
LIN {X 0,Y 481.665,Z 138.485,A -85,B 0,C 180,E1 -6822.157,E2 -6822.157} C_VEL
LIN {X 0,Y 481.725,Z 138.479,A -85,B 0,C 180,E1 -6824.775,E2 -6824.775} C_VEL
LIN {X 0,Y 481.747,Z 138.477,A -85,B 0,C 180,E1 -6828.215,E2 -6828.215} C_VEL
LIN {X 0,Y 481.716,Z 138.476,A -85,B 0,C 180,E1 -6831.611,E2 -6831.611} C_VEL
LIN {X 0,Y 481.768,Z 138.476,A -85,B 0,C 180,E1 -6834.139,E2 -6834.139} C_VEL
LIN {X 0,Y 481.902,Z 138.454,A -85,B 0,C 180,E1 -6837.492,E2 -6837.492} C_VEL
LIN {X 0,Y 481.906,Z 138.459,A -85,B 0,C 180,E1 -6840,E2 -6840} C_VEL
LIN {X 0,Y 481.901,Z 138.455,A -85,B 0,C 180,E1 -6842.508,E2 -6842.508} C_VEL
LIN {X 0,Y 481.766,Z 138.477,A -85,B 0,C 180,E1 -6845.861,E2 -6845.861} C_VEL
LIN {X 0,Y 481.708,Z 138.479,A -85,B 0,C 180,E1 -6848.389,E2 -6848.389} C_VEL
LIN {X 0,Y 481.721,Z 138.483,A -85,B 0,C 180,E1 -6851.786,E2 -6851.786} C_VEL
LIN {X 0,Y 481.686,Z 138.482,A -85,B 0,C 180,E1 -6855.226,E2 -6855.226} C_VEL
LIN {X 0,Y 481.645,Z 138.485,A -85,B 0,C 180,E1 -6858.724,E2 -6858.724} C_VEL
LIN {X 0,Y 481.626,Z 138.494,A -85,B 0,C 180,E1 -6861.396,E2 -6861.396} C_VEL
LIN {X 0,Y 481.638,Z 138.486,A -85,B 0,C 180,E1 -6864.115,E2 -6864.115} C_VEL
LIN {X 0,Y 481.647,Z 138.49,A -85,B 0,C 180,E1 -6867.117,E2 -6867.117} C_VEL
LIN {X 0,Y 481.596,Z 138.493,A -85,B 0,C 180,E1 -6869.747,E2 -6869.747} C_VEL
LIN {X 0,Y 481.647,Z 138.487,A -85,B 0,C 180,E1 -6872.676,E2 -6872.676} C_VEL
LIN {X 0,Y 481.626,Z 138.488,A -85,B 0,C 180,E1 -6875.711,E2 -6875.711} C_VEL
LIN {X 0,Y 481.664,Z 138.489,A -85,B 0,C 180,E1 -6878.86,E2 -6878.86} C_VEL
LIN {X 0,Y 481.614,Z 138.489,A -85,B 0,C 180,E1 -6882.165,E2 -6882.165} C_VEL
LIN {X 0,Y 481.653,Z 138.487,A -85,B 0,C 180,E1 -6884.458,E2 -6884.458} C_VEL
LIN {X 0,Y 481.615,Z 138.495,A -85,B 0,C 180,E1 -6886.855,E2 -6886.855} C_VEL
LIN {X 0,Y 481.657,Z 138.484,A -85,B 0,C 180,E1 -6890.058,E2 -6890.058} C_VEL
LIN {X 0,Y 481.62,Z 138.489,A -85,B 0,C 180,E1 -6893.253,E2 -6893.253} C_VEL
LIN {X 0,Y 481.671,Z 138.488,A -85,B 0,C 180,E1 -6896.327,E2 -6896.327} C_VEL
LIN {X 0,Y 481.647,Z 138.487,A -85,B 0,C 180,E1 -6899.419,E2 -6899.419} C_VEL
LIN {X 0,Y 481.653,Z 138.491,A -85,B 0,C 180,E1 -6902.165,E2 -6902.165} C_VEL
LIN {X 0,Y 481.683,Z 138.585,A -85,B 0,C 180,E1 -6904.376,E2 -6904.376} C_VEL
LIN {X 0,Y 483.664,Z 148.885,A -85,B 0,C 180,E1 -6906.268,E2 -6906.268} C_VEL
LIN {X 0,Y 483.266,Z 163.031,A -85,B 0,C 180,E1 -6908.68,E2 -6908.68} C_VEL
LIN {X 0,Y 482.535,Z 182.64,A -85,B 0,C 180,E1 -6911.971,E2 -6911.971} C_VEL
LIN {X 0,Y 482.246,Z 191.655,A -85,B 0,C 180,E1 -6913.471,E2 -6913.471} C_VEL
LIN {X 0,Y 484.832,Z 210.024,A -85,B 0,C 180,E1 -6913.849,E2 -6913.849} C_VEL
LIN {X 0,Y 484.229,Z 300.115,A -85,B 0,C 180,E1 -6915.205,E2 -6915.205} C_VEL
LIN {X 0,Y 483.905,Z 313.396,A -85,B 0,C 180,E1 -6915.571,E2 -6915.571} C_VEL
LIN {X 0,Y 483.542,Z 325.57,A -85,B 0,C 180,E1 -6916.07,E2 -6916.07} C_VEL
LIN {X 0,Y 483.1,Z 336.34,A -85,B 0,C 180,E1 -6916.658,E2 -6916.658} C_VEL
LIN {X 0,Y 482.629,Z 348.117,A -85,B 0,C 180,E1 -6917.486,E2 -6917.486} C_VEL
LIN {X 0,Y 482.229,Z 358.85,A -85,B 0,C 180,E1 -6918.44,E2 -6918.44} C_VEL
LIN {X 0,Y 481.778,Z 368.474,A -85,B 0,C 180,E1 -6919.493,E2 -6919.493} C_VEL
LIN {X 0,Y 481.462,Z 376.367,A -85,B 0,C 180,E1 -6920.548,E2 -6920.548} C_VEL
LIN {X 0,Y 481.173,Z 384.077,A -85,B 0,C 180,E1 -6921.812,E2 -6921.812} C_VEL
LIN {X 0,Y 481.016,Z 389.362,A -85,B 0,C 180,E1 -6922.866,E2 -6922.866} C_VEL
LIN {X 0,Y 480.91,Z 394.484,A -85,B 0,C 180,E1 -6924.128,E2 -6924.128} C_VEL
LIN {X 0,Y 480.837,Z 398.461,A -85,B 0,C 180,E1 -6925.389,E2 -6925.389} C_VEL
LIN {X 0,Y 480.888,Z 401.403,A -85,B 0,C 180,E1 -6926.648,E2 -6926.648} C_VEL
LIN {X 0,Y 480.821,Z 403.798,A -85,B 0,C 180,E1 -6928.324,E2 -6928.324} C_VEL
LIN {X 0,Y 480.75,Z 404.622,A -85,B 0,C 180,E1 -6930,E2 -6930} C_VEL
LIN {X 0,Y 480.821,Z 403.8,A -85,B 0,C 180,E1 -6931.675,E2 -6931.675} C_VEL
LIN {X 0,Y 480.888,Z 401.407,A -85,B 0,C 180,E1 -6933.351,E2 -6933.351} C_VEL
LIN {X 0,Y 480.836,Z 398.463,A -85,B 0,C 180,E1 -6934.61,E2 -6934.61} C_VEL
LIN {X 0,Y 480.914,Z 394.483,A -85,B 0,C 180,E1 -6935.871,E2 -6935.871} C_VEL
LIN {X 0,Y 481.101,Z 388.365,A -85,B 0,C 180,E1 -6937.343,E2 -6937.343} C_VEL
LIN {X 0,Y 481.296,Z 381.677,A -85,B 0,C 180,E1 -6938.607,E2 -6938.607} C_VEL
LIN {X 0,Y 481.579,Z 373.381,A -85,B 0,C 180,E1 -6939.873,E2 -6939.873} C_VEL
LIN {X 0,Y 481.96,Z 364.883,A -85,B 0,C 180,E1 -6940.927,E2 -6940.927} C_VEL
LIN {X 0,Y 482.397,Z 354.439,A -85,B 0,C 180,E1 -6941.976,E2 -6941.976} C_VEL
LIN {X 0,Y 482.862,Z 342.715,A -85,B 0,C 180,E1 -6942.92,E2 -6942.92} C_VEL
LIN {X 0,Y 483.309,Z 330.692,A -85,B 0,C 180,E1 -6943.667,E2 -6943.667} C_VEL
LIN {X 0,Y 483.728,Z 318.34,A -85,B 0,C 180,E1 -6944.245,E2 -6944.245} C_VEL
LIN {X 0,Y 484.129,Z 305.672,A -85,B 0,C 180,E1 -6944.663,E2 -6944.663} C_VEL
LIN {X 0,Y 484.333,Z 292.451,A -85,B 0,C 180,E1 -6944.925,E2 -6944.925} C_VEL
LIN {X 0,Y 484.692,Z 207.717,A -85,B 0,C 180,E1 -6946.189,E2 -6946.189} C_VEL
LIN {X 0,Y 482.232,Z 191.598,A -85,B 0,C 180,E1 -6946.537,E2 -6946.537} C_VEL
LIN {X 0,Y 482.788,Z 174.74,A -85,B 0,C 180,E1 -6949.349,E2 -6949.349} C_VEL
LIN {X 0,Y 483.525,Z 156.469,A -85,B 0,C 180,E1 -6952.428,E2 -6952.428} C_VEL
LIN {X 0,Y 483.681,Z 148.836,A -85,B 0,C 180,E1 -6953.736,E2 -6953.736} C_VEL
LIN {X 0,Y 481.688,Z 138.487,A -85,B 0,C 180,E1 -6955.671,E2 -6955.671} C_VEL
LIN {X 0,Y 481.658,Z 138.486,A -85,B 0,C 180,E1 -6958.783,E2 -6958.783} C_VEL
LIN {X 0,Y 481.64,Z 138.492,A -85,B 0,C 180,E1 -6961.688,E2 -6961.688} C_VEL
LIN {X 0,Y 481.678,Z 138.481,A -85,B 0,C 180,E1 -6964.682,E2 -6964.682} C_VEL
LIN {X 0,Y 481.645,Z 138.486,A -85,B 0,C 180,E1 -6968.005,E2 -6968.005} C_VEL
LIN {X 0,Y 481.626,Z 138.491,A -85,B 0,C 180,E1 -6971.044,E2 -6971.044} C_VEL
LIN {X 0,Y 481.648,Z 138.485,A -85,B 0,C 180,E1 -6974.457,E2 -6974.457} C_VEL
LIN {X 0,Y 481.617,Z 138.489,A -85,B 0,C 180,E1 -6977.836,E2 -6977.836} C_VEL
LIN {X 0,Y 481.658,Z 138.49,A -85,B 0,C 180,E1 -6981.14,E2 -6981.14} C_VEL
LIN {X 0,Y 481.649,Z 138.49,A -85,B 0,C 180,E1 -6984.796,E2 -6984.796} C_VEL
LIN {X 0,Y 481.639,Z 138.485,A -85,B 0,C 180,E1 -6987.812,E2 -6987.812} C_VEL
LIN {X 0,Y 481.63,Z 138.49,A -85,B 0,C 180,E1 -6991.105,E2 -6991.105} C_VEL
LIN {X 0,Y 481.633,Z 138.487,A -85,B 0,C 180,E1 -6994.039,E2 -6994.039} C_VEL
LIN {X 0,Y 481.642,Z 138.49,A -85,B 0,C 180,E1 -6996.818,E2 -6996.818} C_VEL
LIN {X 0,Y 481.669,Z 138.482,A -85,B 0,C 180,E1 -6999.502,E2 -6999.502} C_VEL
LIN {X 0,Y 481.652,Z 138.488,A -85,B 0,C 180,E1 -7002.156,E2 -7002.156} C_VEL
LIN {X 0,Y 481.718,Z 138.479,A -85,B 0,C 180,E1 -7004.775,E2 -7004.775} C_VEL
LIN {X 0,Y 481.724,Z 138.482,A -85,B 0,C 180,E1 -7008.214,E2 -7008.214} C_VEL
LIN {X 0,Y 481.704,Z 138.479,A -85,B 0,C 180,E1 -7011.611,E2 -7011.611} C_VEL
LIN {X 0,Y 481.76,Z 138.479,A -85,B 0,C 180,E1 -7014.139,E2 -7014.139} C_VEL
LIN {X 0,Y 481.895,Z 138.455,A -85,B 0,C 180,E1 -7017.492,E2 -7017.492} C_VEL
LIN {X 0,Y 481.899,Z 138.461,A -85,B 0,C 180,E1 -7020,E2 -7020} C_VEL
LIN {X 0,Y 481.896,Z 138.455,A -85,B 0,C 180,E1 -7022.508,E2 -7022.508} C_VEL
LIN {X 0,Y 481.766,Z 138.477,A -85,B 0,C 180,E1 -7025.861,E2 -7025.861} C_VEL
LIN {X 0,Y 481.724,Z 138.476,A -85,B 0,C 180,E1 -7028.389,E2 -7028.389} C_VEL
LIN {X 0,Y 481.74,Z 138.479,A -85,B 0,C 180,E1 -7031.785,E2 -7031.785} C_VEL
LIN {X 0,Y 481.718,Z 138.479,A -85,B 0,C 180,E1 -7035.225,E2 -7035.225} C_VEL
LIN {X 0,Y 481.695,Z 138.479,A -85,B 0,C 180,E1 -7038.723,E2 -7038.723} C_VEL
LIN {X 0,Y 481.636,Z 138.494,A -85,B 0,C 180,E1 -7041.395,E2 -7041.395} C_VEL
LIN {X 0,Y 481.638,Z 138.486,A -85,B 0,C 180,E1 -7044.115,E2 -7044.115} C_VEL
LIN {X 0,Y 481.663,Z 138.49,A -85,B 0,C 180,E1 -7047.122,E2 -7047.122} C_VEL
LIN {X 0,Y 481.657,Z 138.484,A -85,B 0,C 180,E1 -7049.743,E2 -7049.743} C_VEL
LIN {X 0,Y 481.644,Z 138.488,A -85,B 0,C 180,E1 -7052.676,E2 -7052.676} C_VEL
LIN {X 0,Y 481.628,Z 138.487,A -85,B 0,C 180,E1 -7055.71,E2 -7055.71} C_VEL
LIN {X 0,Y 481.659,Z 138.491,A -85,B 0,C 180,E1 -7058.86,E2 -7058.86} C_VEL
LIN {X 0,Y 481.619,Z 138.489,A -85,B 0,C 180,E1 -7062.164,E2 -7062.164} C_VEL
LIN {X 0,Y 481.649,Z 138.484,A -85,B 0,C 180,E1 -7065.543,E2 -7065.543} C_VEL
LIN {X 0,Y 481.643,Z 138.488,A -85,B 0,C 180,E1 -7068.958,E2 -7068.958} C_VEL
LIN {X 0,Y 481.646,Z 138.486,A -85,B 0,C 180,E1 -7071.995,E2 -7071.995} C_VEL
LIN {X 0,Y 481.685,Z 138.48,A -85,B 0,C 180,E1 -7075.319,E2 -7075.319} C_VEL
LIN {X 0,Y 481.642,Z 138.493,A -85,B 0,C 180,E1 -7078.312,E2 -7078.312} C_VEL
LIN {X 0,Y 481.659,Z 138.483,A -85,B 0,C 180,E1 -7081.217,E2 -7081.217} C_VEL
LIN {X 0,Y 481.659,Z 138.489,A -85,B 0,C 180,E1 -7084.041,E2 -7084.041} C_VEL
LIN {X 0,Y 481.674,Z 138.482,A -85,B 0,C 180,E1 -7086.813,E2 -7086.813} C_VEL
LIN {X 0,Y 481.636,Z 138.489,A -85,B 0,C 180,E1 -7087.94,E2 -7087.94} C_VEL
LIN {X 0,Y 480.994,Z 138.721,A -85,B 0,C 180,E1 -7088.413,E2 -7088.413} C_VEL
LIN {X 0,Y 478.376,Z 139.978,A -85,B 0,C 180,E1 -7089.149,E2 -7089.149} C_VEL
LIN {X 0,Y 475.923,Z 142.241,A -85,B 0,C 180,E1 -7089.861,E2 -7089.861} C_VEL
LIN {X 0,Y 475.543,Z 144.063,A -85,B 0,C 180,E1 -7090.291,E2 -7090.291} C_VEL
LIN {X 0,Y 475.709,Z 147.639,A -85,B 0,C 180,E1 -7091.034,E2 -7091.034} C_VEL
LIN {X 0,Y 475.449,Z 159.137,A -85,B 0,C 180,E1 -7093.302,E2 -7093.302} C_VEL
LIN {X 0,Y 478.184,Z 172.862,A -85,B 0,C 180,E1 -7093.613,E2 -7093.613} C_VEL
LIN {X 0,Y 477.537,Z 266.541,A -85,B 0,C 180,E1 -7095.049,E2 -7095.049} C_VEL
LIN {X 0,Y 477.265,Z 279.657,A -85,B 0,C 180,E1 -7095.422,E2 -7095.422} C_VEL
LIN {X 0,Y 476.908,Z 291.719,A -85,B 0,C 180,E1 -7095.928,E2 -7095.928} C_VEL
LIN {X 0,Y 476.531,Z 302.82,A -85,B 0,C 180,E1 -7096.552,E2 -7096.552} C_VEL
LIN {X 0,Y 476.218,Z 313.463,A -85,B 0,C 180,E1 -7097.32,E2 -7097.32} C_VEL
LIN {X 0,Y 475.656,Z 324.146,A -85,B 0,C 180,E1 -7098.279,E2 -7098.279} C_VEL
LIN {X 0,Y 475.26,Z 333.752,A -85,B 0,C 180,E1 -7099.348,E2 -7099.348} C_VEL
LIN {X 0,Y 474.84,Z 341.621,A -85,B 0,C 180,E1 -7100.416,E2 -7100.416} C_VEL
LIN {X 0,Y 474.456,Z 349.312,A -85,B 0,C 180,E1 -7101.697,E2 -7101.697} C_VEL
LIN {X 0,Y 474.187,Z 356.364,A -85,B 0,C 180,E1 -7103.191,E2 -7103.191} C_VEL
LIN {X 0,Y 473.988,Z 361.064,A -85,B 0,C 180,E1 -7104.47,E2 -7104.47} C_VEL
LIN {X 0,Y 473.936,Z 364.659,A -85,B 0,C 180,E1 -7105.748,E2 -7105.748} C_VEL
LIN {X 0,Y 473.886,Z 366.518,A -85,B 0,C 180,E1 -7106.6,E2 -7106.6} C_VEL
LIN {X 0,Y 473.799,Z 367.922,A -85,B 0,C 180,E1 -7107.45,E2 -7107.45} C_VEL
LIN {X 0,Y 473.695,Z 369.535,A -85,B 0,C 180,E1 -7109.15,E2 -7109.15} C_VEL
LIN {X 0,Y 473.679,Z 369.771,A -85,B 0,C 180,E1 -7110,E2 -7110} C_VEL
LIN {X 0,Y 473.695,Z 369.585,A -85,B 0,C 180,E1 -7110.851,E2 -7110.851} C_VEL
LIN {X 0,Y 473.761,Z 369.001,A -85,B 0,C 180,E1 -7111.701,E2 -7111.701} C_VEL
LIN {X 0,Y 473.886,Z 366.684,A -85,B 0,C 180,E1 -7113.401,E2 -7113.401} C_VEL
LIN {X 0,Y 473.91,Z 363.828,A -85,B 0,C 180,E1 -7114.679,E2 -7114.679} C_VEL
LIN {X 0,Y 474.118,Z 359.949,A -85,B 0,C 180,E1 -7115.956,E2 -7115.956} C_VEL
LIN {X 0,Y 474.22,Z 354.95,A -85,B 0,C 180,E1 -7117.237,E2 -7117.237} C_VEL
LIN {X 0,Y 474.528,Z 348.653,A -85,B 0,C 180,E1 -7118.517,E2 -7118.517} C_VEL
LIN {X 0,Y 474.877,Z 340.768,A -85,B 0,C 180,E1 -7119.799,E2 -7119.799} C_VEL
LIN {X 0,Y 475.232,Z 332.729,A -85,B 0,C 180,E1 -7120.869,E2 -7120.869} C_VEL
LIN {X 0,Y 475.752,Z 322.913,A -85,B 0,C 180,E1 -7121.936,E2 -7121.936} C_VEL
LIN {X 0,Y 476.219,Z 311.782,A -85,B 0,C 180,E1 -7122.906,E2 -7122.906} C_VEL
LIN {X 0,Y 476.682,Z 299.299,A -85,B 0,C 180,E1 -7123.753,E2 -7123.753} C_VEL
LIN {X 0,Y 477.077,Z 287.978,A -85,B 0,C 180,E1 -7124.34,E2 -7124.34} C_VEL
LIN {X 0,Y 477.391,Z 275.09,A -85,B 0,C 180,E1 -7124.821,E2 -7124.821} C_VEL
LIN {X 0,Y 477.659,Z 261.332,A -85,B 0,C 180,E1 -7125.139,E2 -7125.139} C_VEL
LIN {X 0,Y 478.086,Z 172.58,A -85,B 0,C 180,E1 -7126.487,E2 -7126.487} C_VEL
LIN {X 0,Y 475.437,Z 158.984,A -85,B 0,C 180,E1 -7126.798,E2 -7126.798} C_VEL
LIN {X 0,Y 475.819,Z 146.12,A -85,B 0,C 180,E1 -7129.366,E2 -7129.366} C_VEL
LIN {X 0,Y 474.697,Z 139.356,A -85,B 0,C 180,E1 -7130.864,E2 -7130.864} C_VEL
LIN {X 0,Y 474.63,Z 139.361,A -85,B 0,C 180,E1 -7134.495,E2 -7134.495} C_VEL
LIN {X 0,Y 474.639,Z 139.359,A -85,B 0,C 180,E1 -7137.324,E2 -7137.324} C_VEL
LIN {X 0,Y 474.603,Z 139.364,A -85,B 0,C 180,E1 -7140.23,E2 -7140.23} C_VEL
LIN {X 0,Y 474.645,Z 139.359,A -85,B 0,C 180,E1 -7143.22,E2 -7143.22} C_VEL
LIN {X 0,Y 474.585,Z 139.365,A -85,B 0,C 180,E1 -7146.324,E2 -7146.324} C_VEL
LIN {X 0,Y 474.622,Z 139.367,A -85,B 0,C 180,E1 -7149.548,E2 -7149.548} C_VEL
LIN {X 0,Y 474.598,Z 139.363,A -85,B 0,C 180,E1 -7152.233,E2 -7152.233} C_VEL
LIN {X 0,Y 474.616,Z 139.368,A -85,B 0,C 180,E1 -7155.298,E2 -7155.298} C_VEL
LIN {X 0,Y 474.608,Z 139.361,A -85,B 0,C 180,E1 -7158.213,E2 -7158.213} C_VEL
LIN {X 0,Y 474.607,Z 139.365,A -85,B 0,C 180,E1 -7161.542,E2 -7161.542} C_VEL
LIN {X 0,Y 474.618,Z 139.363,A -85,B 0,C 180,E1 -7164.725,E2 -7164.725} C_VEL
LIN {X 0,Y 474.624,Z 139.36,A -85,B 0,C 180,E1 -7167.787,E2 -7167.787} C_VEL
LIN {X 0,Y 474.596,Z 139.371,A -85,B 0,C 180,E1 -7170.89,E2 -7170.89} C_VEL
LIN {X 0,Y 474.608,Z 139.362,A -85,B 0,C 180,E1 -7173.625,E2 -7173.625} C_VEL
LIN {X 0,Y 474.632,Z 139.365,A -85,B 0,C 180,E1 -7176.642,E2 -7176.642} C_VEL
LIN {X 0,Y 474.645,Z 139.358,A -85,B 0,C 180,E1 -7180.089,E2 -7180.089} C_VEL
LIN {X 0,Y 474.589,Z 139.369,A -85,B 0,C 180,E1 -7182.772,E2 -7182.772} C_VEL
LIN {X 0,Y 474.628,Z 139.359,A -85,B 0,C 180,E1 -7185.42,E2 -7185.42} C_VEL
LIN {X 0,Y 474.701,Z 139.353,A -85,B 0,C 180,E1 -7188.037,E2 -7188.037} C_VEL
LIN {X 0,Y 474.692,Z 139.351,A -85,B 0,C 180,E1 -7191.486,E2 -7191.486} C_VEL
LIN {X 0,Y 474.731,Z 139.351,A -85,B 0,C 180,E1 -7194.052,E2 -7194.052} C_VEL
LIN {X 0,Y 474.867,Z 139.33,A -85,B 0,C 180,E1 -7197.455,E2 -7197.455} C_VEL
LIN {X 0,Y 474.875,Z 139.335,A -85,B 0,C 180,E1 -7200,E2 -7200} C_VEL
LIN {X 0,Y 474.866,Z 139.331,A -85,B 0,C 180,E1 -7202.545,E2 -7202.545} C_VEL
LIN {X 0,Y 474.729,Z 139.354,A -85,B 0,C 180,E1 -7205.948,E2 -7205.948} C_VEL
LIN {X 0,Y 474.656,Z 139.356,A -85,B 0,C 180,E1 -7208.515,E2 -7208.515} C_VEL
LIN {X 0,Y 474.68,Z 139.357,A -85,B 0,C 180,E1 -7211.963,E2 -7211.963} C_VEL
LIN {X 0,Y 474.646,Z 139.362,A -85,B 0,C 180,E1 -7215.457,E2 -7215.457} C_VEL
LIN {X 0,Y 474.6,Z 139.364,A -85,B 0,C 180,E1 -7219.013,E2 -7219.013} C_VEL
LIN {X 0,Y 474.571,Z 139.37,A -85,B 0,C 180,E1 -7221.73,E2 -7221.73} C_VEL
LIN {X 0,Y 474.618,Z 139.36,A -85,B 0,C 180,E1 -7224.495,E2 -7224.495} C_VEL
LIN {X 0,Y 474.593,Z 139.371,A -85,B 0,C 180,E1 -7227.327,E2 -7227.327} C_VEL
LIN {X 0,Y 474.546,Z 139.369,A -85,B 0,C 180,E1 -7230.234,E2 -7230.234} C_VEL
LIN {X 0,Y 474.611,Z 139.368,A -85,B 0,C 180,E1 -7233.223,E2 -7233.223} C_VEL
LIN {X 0,Y 474.58,Z 139.365,A -85,B 0,C 180,E1 -7236.324,E2 -7236.324} C_VEL
LIN {X 0,Y 474.62,Z 139.361,A -85,B 0,C 180,E1 -7239.548,E2 -7239.548} C_VEL
LIN {X 0,Y 474.575,Z 139.366,A -85,B 0,C 180,E1 -7242.23,E2 -7242.23} C_VEL
LIN {X 0,Y 474.615,Z 139.362,A -85,B 0,C 180,E1 -7245.298,E2 -7245.298} C_VEL
LIN {X 0,Y 474.591,Z 139.365,A -85,B 0,C 180,E1 -7248.212,E2 -7248.212} C_VEL
LIN {X 0,Y 474.608,Z 139.361,A -85,B 0,C 180,E1 -7251.542,E2 -7251.542} C_VEL
LIN {X 0,Y 474.62,Z 139.365,A -85,B 0,C 180,E1 -7254.725,E2 -7254.725} C_VEL
LIN {X 0,Y 474.628,Z 139.36,A -85,B 0,C 180,E1 -7257.787,E2 -7257.787} C_VEL
LIN {X 0,Y 474.6,Z 139.366,A -85,B 0,C 180,E1 -7260.89,E2 -7260.89} C_VEL
LIN {X 0,Y 474.6,Z 139.369,A -85,B 0,C 180,E1 -7263.625,E2 -7263.625} C_VEL
LIN {X 0,Y 474.651,Z 139.425,A -85,B 0,C 180,E1 -7264.166,E2 -7264.166} C_VEL
LIN {X 0,Y 476.74,Z 150.454,A -85,B 0,C 180,E1 -7266.223,E2 -7266.223} C_VEL
LIN {X 0,Y 476.342,Z 163.52,A -85,B 0,C 180,E1 -7268.484,E2 -7268.484} C_VEL
LIN {X 0,Y 475.511,Z 183.685,A -85,B 0,C 180,E1 -7271.918,E2 -7271.918} C_VEL
LIN {X 0,Y 475.26,Z 191.444,A -85,B 0,C 180,E1 -7273.229,E2 -7273.229} C_VEL
LIN {X 0,Y 478.015,Z 210.767,A -85,B 0,C 180,E1 -7273.628,E2 -7273.628} C_VEL
LIN {X 0,Y 477.375,Z 299.866,A -85,B 0,C 180,E1 -7274.988,E2 -7274.988} C_VEL
LIN {X 0,Y 477.029,Z 313.144,A -85,B 0,C 180,E1 -7275.359,E2 -7275.359} C_VEL
LIN {X 0,Y 476.629,Z 325.315,A -85,B 0,C 180,E1 -7275.864,E2 -7275.864} C_VEL
LIN {X 0,Y 476.115,Z 337.6,A -85,B 0,C 180,E1 -7276.556,E2 -7276.556} C_VEL
LIN {X 0,Y 475.632,Z 348.791,A -85,B 0,C 180,E1 -7277.376,E2 -7277.376} C_VEL
LIN {X 0,Y 475.197,Z 359.666,A -85,B 0,C 180,E1 -7278.375,E2 -7278.375} C_VEL
LIN {X 0,Y 474.749,Z 368.215,A -85,B 0,C 180,E1 -7279.336,E2 -7279.336} C_VEL
LIN {X 0,Y 474.436,Z 376.108,A -85,B 0,C 180,E1 -7280.407,E2 -7280.407} C_VEL
LIN {X 0,Y 474.129,Z 383.818,A -85,B 0,C 180,E1 -7281.69,E2 -7281.69} C_VEL
LIN {X 0,Y 473.896,Z 390.928,A -85,B 0,C 180,E1 -7283.186,E2 -7283.186} C_VEL
LIN {X 0,Y 473.836,Z 395.661,A -85,B 0,C 180,E1 -7284.467,E2 -7284.467} C_VEL
LIN {X 0,Y 473.733,Z 399.275,A -85,B 0,C 180,E1 -7285.746,E2 -7285.746} C_VEL
LIN {X 0,Y 473.795,Z 401.144,A -85,B 0,C 180,E1 -7286.598,E2 -7286.598} C_VEL
LIN {X 0,Y 473.724,Z 403.539,A -85,B 0,C 180,E1 -7288.299,E2 -7288.299} C_VEL
LIN {X 0,Y 473.692,Z 404.147,A -85,B 0,C 180,E1 -7289.149,E2 -7289.149} C_VEL
LIN {X 0,Y 473.676,Z 404.364,A -85,B 0,C 180,E1 -7290,E2 -7290} C_VEL
LIN {X 0,Y 473.692,Z 404.148,A -85,B 0,C 180,E1 -7290.85,E2 -7290.85} C_VEL
LIN {X 0,Y 473.724,Z 403.541,A -85,B 0,C 180,E1 -7291.7,E2 -7291.7} C_VEL
LIN {X 0,Y 473.795,Z 401.147,A -85,B 0,C 180,E1 -7293.401,E2 -7293.401} C_VEL
LIN {X 0,Y 473.76,Z 398.204,A -85,B 0,C 180,E1 -7294.679,E2 -7294.679} C_VEL
LIN {X 0,Y 473.822,Z 394.222,A -85,B 0,C 180,E1 -7295.959,E2 -7295.959} C_VEL
LIN {X 0,Y 474.011,Z 388.103,A -85,B 0,C 180,E1 -7297.454,E2 -7297.454} C_VEL
LIN {X 0,Y 474.244,Z 381.415,A -85,B 0,C 180,E1 -7298.736,E2 -7298.736} C_VEL
LIN {X 0,Y 474.54,Z 373.119,A -85,B 0,C 180,E1 -7300.021,E2 -7300.021} C_VEL
LIN {X 0,Y 474.963,Z 364.621,A -85,B 0,C 180,E1 -7301.09,E2 -7301.09} C_VEL
LIN {X 0,Y 475.413,Z 354.39,A -85,B 0,C 180,E1 -7302.135,E2 -7302.135} C_VEL
LIN {X 0,Y 475.856,Z 344.024,A -85,B 0,C 180,E1 -7302.994,E2 -7302.994} C_VEL
LIN {X 0,Y 476.325,Z 332.352,A -85,B 0,C 180,E1 -7303.763,E2 -7303.763} C_VEL
LIN {X 0,Y 476.751,Z 320.68,A -85,B 0,C 180,E1 -7304.349,E2 -7304.349} C_VEL
LIN {X 0,Y 477.213,Z 307.236,A -85,B 0,C 180,E1 -7304.825,E2 -7304.825} C_VEL
LIN {X 0,Y 477.483,Z 293.954,A -85,B 0,C 180,E1 -7305.117,E2 -7305.117} C_VEL
LIN {X 0,Y 477.881,Z 208.716,A -85,B 0,C 180,E1 -7306.406,E2 -7306.406} C_VEL
LIN {X 0,Y 475.257,Z 191.404,A -85,B 0,C 180,E1 -7306.775,E2 -7306.775} C_VEL
LIN {X 0,Y 475.824,Z 174.665,A -85,B 0,C 180,E1 -7309.611,E2 -7309.611} C_VEL
LIN {X 0,Y 476.592,Z 157.522,A -85,B 0,C 180,E1 -7312.544,E2 -7312.544} C_VEL
LIN {X 0,Y 476.661,Z 149.667,A -85,B 0,C 180,E1 -7313.915,E2 -7313.915} C_VEL
LIN {X 0,Y 474.648,Z 139.364,A -85,B 0,C 180,E1 -7315.866,E2 -7315.866} C_VEL
LIN {X 0,Y 474.597,Z 139.368,A -85,B 0,C 180,E1 -7319.109,E2 -7319.109} C_VEL
LIN {X 0,Y 474.599,Z 139.363,A -85,B 0,C 180,E1 -7322.427,E2 -7322.427} C_VEL
LIN {X 0,Y 474.605,Z 139.37,A -85,B 0,C 180,E1 -7325.467,E2 -7325.467} C_VEL
LIN {X 0,Y 474.604,Z 139.362,A -85,B 0,C 180,E1 -7328.457,E2 -7328.457} C_VEL
LIN {X 0,Y 474.598,Z 139.365,A -85,B 0,C 180,E1 -7331.786,E2 -7331.786} C_VEL
LIN {X 0,Y 474.61,Z 139.363,A -85,B 0,C 180,E1 -7334.701,E2 -7334.701} C_VEL
LIN {X 0,Y 474.577,Z 139.366,A -85,B 0,C 180,E1 -7337.768,E2 -7337.768} C_VEL
LIN {X 0,Y 474.614,Z 139.362,A -85,B 0,C 180,E1 -7340.451,E2 -7340.451} C_VEL
LIN {X 0,Y 474.576,Z 139.366,A -85,B 0,C 180,E1 -7343.675,E2 -7343.675} C_VEL
LIN {X 0,Y 474.606,Z 139.368,A -85,B 0,C 180,E1 -7346.777,E2 -7346.777} C_VEL
LIN {X 0,Y 474.586,Z 139.364,A -85,B 0,C 180,E1 -7349.768,E2 -7349.768} C_VEL
LIN {X 0,Y 474.593,Z 139.371,A -85,B 0,C 180,E1 -7352.684,E2 -7352.684} C_VEL
LIN {X 0,Y 474.616,Z 139.36,A -85,B 0,C 180,E1 -7355.505,E2 -7355.505} C_VEL
LIN {X 0,Y 474.614,Z 139.364,A -85,B 0,C 180,E1 -7358.887,E2 -7358.887} C_VEL
LIN {X 0,Y 474.619,Z 139.361,A -85,B 0,C 180,E1 -7361.883,E2 -7361.883} C_VEL
LIN {X 0,Y 474.677,Z 139.359,A -85,B 0,C 180,E1 -7364.544,E2 -7364.544} C_VEL
LIN {X 0,Y 474.682,Z 139.357,A -85,B 0,C 180,E1 -7368.037,E2 -7368.037} C_VEL
LIN {X 0,Y 474.653,Z 139.356,A -85,B 0,C 180,E1 -7371.485,E2 -7371.485} C_VEL
LIN {X 0,Y 474.724,Z 139.354,A -85,B 0,C 180,E1 -7374.052,E2 -7374.052} C_VEL
LIN {X 0,Y 474.86,Z 139.331,A -85,B 0,C 180,E1 -7377.455,E2 -7377.455} C_VEL
LIN {X 0,Y 474.868,Z 139.337,A -85,B 0,C 180,E1 -7380,E2 -7380} C_VEL
LIN {X 0,Y 474.861,Z 139.331,A -85,B 0,C 180,E1 -7382.545,E2 -7382.545} C_VEL
LIN {X 0,Y 474.729,Z 139.352,A -85,B 0,C 180,E1 -7385.948,E2 -7385.948} C_VEL
LIN {X 0,Y 474.697,Z 139.351,A -85,B 0,C 180,E1 -7388.514,E2 -7388.514} C_VEL
LIN {X 0,Y 474.694,Z 139.354,A -85,B 0,C 180,E1 -7391.963,E2 -7391.963} C_VEL
